C03651=1231.383,135.058,-50.263,-178.039,5.630,148.402
C03652=1231.378,135.308,-50.283,-178.037,5.631,148.401
C03653=1231.373,135.557,-50.304,-178.035,5.632,148.401
C03654=1231.369,135.806,-50.324,-178.032,5.634,148.400
C03655=1231.363,136.055,-50.345,-178.029,5.634,148.400
C03656=1231.359,136.304,-50.365,-178.027,5.635,148.399
C03657=1231.355,136.553,-50.386,-178.024,5.637,148.399
C03658=1231.349,136.802,-50.407,-178.022,5.638,148.398
C03659=1231.345,137.051,-50.427,-178.019,5.638,148.398
C03660=1231.341,137.300,-50.447,-178.017,5.640,148.397
C03661=1231.335,137.549,-50.468,-178.014,5.641,148.397
C03662=1231.331,137.798,-50.489,-178.011,5.643,148.396
C03663=1231.326,138.048,-50.510,-178.009,5.643,148.395
C03664=1231.321,138.297,-50.530,-178.007,5.644,148.395
C03665=1231.316,138.546,-50.551,-178.004,5.646,148.394
C03666=1231.312,138.795,-50.572,-178.001,5.647,148.394
C03667=1231.307,139.044,-50.592,-177.999,5.647,148.393
C03668=1231.302,139.293,-50.613,-177.996,5.649,148.393
C03669=1231.298,139.542,-50.633,-177.994,5.650,148.392
C03670=1231.293,139.791,-50.654,-177.991,5.651,148.392
C03671=1231.288,140.040,-50.675,-177.988,5.652,148.391
C03672=1231.283,140.289,-50.696,-177.986,5.653,148.391
C03673=1231.279,140.539,-50.716,-177.984,5.654,148.390
C03674=1231.274,140.788,-50.737,-177.981,5.656,148.390
C03675=1231.269,141.037,-50.758,-177.978,5.656,148.389
C03676=1231.264,141.287,-50.779,-177.976,5.657,148.389
C03677=1231.260,141.535,-50.800,-177.973,5.659,148.388
C03678=1231.255,141.784,-50.821,-177.971,5.660,148.388
C03679=1231.251,142.033,-50.841,-177.968,5.661,148.387
C03680=1231.245,142.282,-50.862,-177.966,5.662,148.387
C03681=1231.241,142.531,-50.882,-177.963,5.663,148.386
C03682=1231.236,142.781,-50.903,-177.960,5.665,148.386
C03683=1231.231,143.030,-50.924,-177.958,5.665,148.385
C03684=1231.227,143.279,-50.946,-177.956,5.666,148.385
C03685=1231.223,143.528,-50.966,-177.953,5.668,148.384
C03686=1231.217,143.777,-50.987,-177.950,5.669,148.384
C03687=1231.212,144.026,-51.008,-177.947,5.670,148.383
C03688=1231.208,144.275,-51.028,-177.945,5.671,148.383
C03689=1231.203,144.524,-51.050,-177.943,5.672,148.382
C03690=1231.199,144.773,-51.070,-177.940,5.674,148.382
C03691=1231.193,145.022,-51.091,-177.937,5.674,148.381
C03692=1231.189,145.272,-51.112,-177.935,5.676,148.381
C03693=1231.185,145.520,-51.134,-177.932,5.677,148.380
C03694=1231.179,145.770,-51.155,-177.930,5.678,148.380
C03695=1231.175,146.019,-51.175,-177.927,5.680,148.380
C03696=1231.170,146.267,-51.197,-177.925,5.680,148.379
C03697=1231.165,146.517,-51.218,-177.923,5.681,148.379
C03698=1231.161,146.766,-51.239,-177.919,5.683,148.378
C03699=1231.156,147.015,-51.260,-177.917,5.684,148.378
C03700=1231.152,147.264,-51.281,-177.914,5.685,148.377
C03701=1231.147,147.513,-51.302,-177.912,5.686,148.377
C03702=1231.142,147.762,-51.323,-177.909,5.687,148.376
C03703=1231.137,148.011,-51.344,-177.907,5.689,148.376
C03704=1231.133,148.261,-51.365,-177.904,5.689,148.375
C03705=1231.128,148.509,-51.387,-177.902,5.691,148.375
C03706=1231.123,148.758,-51.408,-177.899,5.692,148.374
C03707=1231.119,149.007,-51.429,-177.896,5.694,148.374
C03708=1231.113,149.256,-51.450,-177.894,5.695,148.373
C03709=1231.109,149.506,-51.471,-177.892,5.695,148.372
C03710=1231.105,149.754,-51.492,-177.889,5.697,148.372
C03711=1231.100,150.004,-51.513,-177.886,5.698,148.372
C03712=1231.095,150.252,-51.535,-177.884,5.700,148.371
C03713=1231.090,150.502,-51.556,-177.881,5.700,148.371
C03714=1231.086,150.751,-51.577,-177.879,5.701,148.370
C03715=1231.081,151.000,-51.598,-177.876,5.703,148.370
C03716=1231.076,151.248,-51.620,-177.874,5.704,148.369
C03717=1231.071,151.498,-51.641,-177.871,5.706,148.369
C03718=1231.067,151.747,-51.662,-177.868,5.706,148.368
C03719=1231.062,151.996,-51.683,-177.866,5.708,148.368
C03720=1231.057,152.245,-51.705,-177.863,5.709,148.367
C03721=1231.052,152.494,-51.726,-177.861,5.710,148.367
C03722=1231.048,152.743,-51.748,-177.858,5.712,148.366
C03723=1231.043,152.992,-51.768,-177.856,5.712,148.366
C03724=1231.038,153.241,-51.790,-177.853,5.714,148.365
C03725=1231.034,153.491,-51.811,-177.851,5.715,148.365
C03726=1231.029,153.739,-51.833,-177.848,5.717,148.364
C03727=1231.024,153.988,-51.855,-177.845,5.717,148.364
C03728=1231.020,154.237,-51.875,-177.843,5.719,148.363
C03729=1231.015,154.486,-51.897,-177.841,5.720,148.363
C03730=1231.010,154.736,-51.918,-177.838,5.721,148.362
C03731=1231.005,154.984,-51.940,-177.835,5.723,148.362
C03732=1231.001,155.234,-51.962,-177.833,5.723,148.361
C03733=1230.996,155.483,-51.983,-177.830,5.725,148.361
C03734=1230.991,155.732,-52.004,-177.828,5.726,148.361
C03735=1230.987,155.981,-52.026,-177.825,5.727,148.360
C03736=1230.982,156.230,-52.047,-177.823,5.728,148.360
C03737=1230.977,156.478,-52.069,-177.820,5.730,148.359
C03738=1230.973,156.728,-52.091,-177.817,5.731,148.359
C03739=1230.968,156.977,-52.112,-177.815,5.732,148.358
C03740=1230.963,157.226,-52.133,-177.812,5.733,148.358
C03741=1230.959,157.475,-52.155,-177.810,5.734,148.357
C03742=1230.954,157.724,-52.177,-177.807,5.736,148.357
C03743=1230.949,157.973,-52.198,-177.805,5.737,148.356
C03744=1230.945,158.222,-52.220,-177.802,5.739,148.356
C03745=1230.940,158.471,-52.242,-177.800,5.739,148.355
C03746=1230.935,158.720,-52.263,-177.797,5.741,148.355
C03747=1230.930,158.970,-52.285,-177.794,5.742,148.354
C03748=1230.925,159.218,-52.306,-177.792,5.744,148.354
C03749=1230.921,159.487,-52.330,-177.790,5.745,148.354
C03750=1230.915,159.756,-52.353,-177.786,5.746,148.353
C03751=1230.910,160.025,-52.377,-177.783,5.748,148.352
C03752=1230.906,160.294,-52.400,-177.781,5.749,148.352
C03753=1230.901,160.543,-52.422,-177.778,5.750,148.351
C03754=1230.896,160.792,-52.443,-177.776,5.751,148.351
C03755=1230.892,161.042,-52.465,-177.773,5.753,148.351
C03756=1230.887,161.290,-52.487,-177.771,5.754,148.350
C03757=1230.882,161.539,-52.508,-177.768,5.756,148.350
C03758=1230.878,161.788,-52.530,-177.766,5.757,148.349
C03759=1230.873,162.037,-52.552,-177.763,5.758,148.349
C03760=1230.869,162.286,-52.574,-177.761,5.759,148.348
C03761=1230.864,162.535,-52.596,-177.758,5.761,148.348
C03762=1230.859,162.785,-52.619,-177.755,5.762,148.347
C03763=1230.854,163.033,-52.640,-177.753,5.763,148.347
C03764=1230.849,163.282,-52.662,-177.750,5.764,148.346
C03765=1230.845,163.531,-52.684,-177.748,5.766,148.346
C03766=1230.840,163.780,-52.706,-177.745,5.767,148.346
C03767=1230.836,164.029,-52.728,-177.742,5.768,148.345
C03768=1230.831,164.278,-52.749,-177.740,5.769,148.345
C03769=1230.827,164.527,-52.771,-177.738,5.771,148.344
C03770=1230.822,164.776,-52.793,-177.735,5.772,148.344
C03771=1230.817,165.025,-52.815,-177.732,5.774,148.343
C03772=1230.813,165.274,-52.837,-177.730,5.774,148.343
C03773=1230.808,165.523,-52.859,-177.727,5.776,148.342
C03774=1230.803,165.772,-52.881,-177.725,5.777,148.342
C03775=1230.798,166.021,-52.903,-177.722,5.779,148.341
C03776=1230.794,166.270,-52.925,-177.720,5.780,148.341
C03777=1230.789,166.519,-52.947,-177.717,5.782,148.340
C03778=1230.784,166.768,-52.969,-177.715,5.782,148.340
C03779=1230.779,167.018,-52.991,-177.712,5.784,148.340
C03780=1230.775,167.266,-53.013,-177.710,5.785,148.339
C03781=1230.770,167.516,-53.035,-177.707,5.787,148.339
C03782=1230.766,167.764,-53.057,-177.705,5.788,148.338
C03783=1230.761,168.013,-53.079,-177.702,5.789,148.338
C03784=1230.756,168.262,-53.102,-177.699,5.791,148.337
C03785=1230.752,168.511,-53.124,-177.697,5.792,148.337
C03786=1230.747,168.760,-53.145,-177.694,5.794,148.336
C03787=1230.742,169.009,-53.167,-177.691,5.794,148.336
C03788=1230.738,169.257,-53.190,-177.689,5.796,148.335
C03789=1230.733,169.507,-53.213,-177.687,5.797,148.335
C03790=1230.728,169.756,-53.234,-177.684,5.799,148.335
C03791=1230.724,170.005,-53.256,-177.681,5.800,148.334
C03792=1230.719,170.254,-53.278,-177.679,5.802,148.334
C03793=1230.714,170.503,-53.301,-177.676,5.802,148.333
C03794=1230.710,170.752,-53.323,-177.674,5.804,148.333
C03795=1230.705,171.001,-53.345,-177.671,5.805,148.332
C03796=1230.700,171.250,-53.368,-177.669,5.807,148.332
C03797=1230.695,171.498,-53.390,-177.666,5.808,148.331
C03798=1230.691,171.748,-53.412,-177.664,5.809,148.331
C03799=1230.686,171.997,-53.434,-177.661,5.811,148.331
C03800=1230.682,172.245,-53.457,-177.658,5.812,148.330
C03801=1230.677,172.495,-53.479,-177.656,5.814,148.330
C03802=1230.672,172.743,-53.501,-177.654,5.815,148.329
C03803=1230.668,172.992,-53.524,-177.650,5.816,148.329
C03804=1230.663,173.241,-53.546,-177.648,5.817,148.328
C03805=1230.658,173.491,-53.569,-177.646,5.819,148.328
C03806=1230.654,173.739,-53.591,-177.643,5.821,148.327
C03807=1230.649,173.988,-53.613,-177.640,5.822,148.327
C03808=1230.644,174.238,-53.636,-177.638,5.823,148.327
C03809=1230.640,174.486,-53.658,-177.636,5.824,148.326
C03810=1230.635,174.735,-53.680,-177.633,5.826,148.326
C03811=1230.631,174.984,-53.703,-177.630,5.827,148.325
C03812=1230.626,175.233,-53.725,-177.628,5.829,148.325
C03813=1230.621,175.482,-53.749,-177.625,5.830,148.324
C03814=1230.617,175.731,-53.771,-177.623,5.831,148.324
C03815=1230.612,175.980,-53.792,-177.620,5.833,148.324
C03816=1230.607,176.229,-53.816,-177.618,5.834,148.323
C03817=1230.603,176.478,-53.838,-177.615,5.836,148.323
C03818=1230.598,176.726,-53.861,-177.613,5.837,148.322
C03819=1230.593,176.976,-53.883,-177.610,5.839,148.322
C03820=1230.589,177.225,-53.906,-177.607,5.840,148.321
C03821=1230.584,177.473,-53.928,-177.605,5.841,148.321
C03822=1230.579,177.722,-53.951,-177.602,5.843,148.321
C03823=1230.575,177.971,-53.974,-177.600,5.844,148.320
C03824=1230.570,178.220,-53.996,-177.597,5.845,148.320
C03825=1230.565,178.469,-54.019,-177.594,5.847,148.319
C03826=1230.561,178.718,-54.041,-177.592,5.848,148.319
C03827=1230.556,178.967,-54.064,-177.589,5.850,148.318
C03828=1230.552,179.216,-54.086,-177.587,5.851,148.318
C03829=1230.547,179.465,-54.109,-177.584,5.853,148.318
C03830=1230.543,179.714,-54.132,-177.582,5.854,148.317
C03831=1230.537,179.963,-54.154,-177.579,5.855,148.317
C03832=1230.533,180.212,-54.178,-177.576,5.857,148.316
C03833=1230.528,180.461,-54.200,-177.574,5.858,148.316
C03834=1230.524,180.710,-54.223,-177.572,5.860,148.316
C03835=1230.519,180.958,-54.246,-177.569,5.861,148.315
C03836=1230.514,181.208,-54.268,-177.566,5.862,148.315
C03837=1230.510,181.456,-54.291,-177.564,5.864,148.314
C03838=1230.505,181.705,-54.314,-177.562,5.865,148.314
C03839=1230.501,181.953,-54.337,-177.559,5.867,148.313
C03840=1230.496,182.203,-54.359,-177.556,5.869,148.313
C03841=1230.491,182.452,-54.383,-177.554,5.870,148.313
C03842=1230.487,182.701,-54.405,-177.551,5.871,148.312
C03843=1230.482,182.950,-54.428,-177.548,5.873,148.312
C03844=1230.478,183.198,-54.451,-177.546,5.874,148.311
C03845=1230.473,183.447,-54.474,-177.543,5.876,148.311
C03846=1230.468,183.697,-54.497,-177.541,5.877,148.311
C03847=1230.464,183.945,-54.520,-177.538,5.878,148.310
C03848=1230.459,184.194,-54.542,-177.535,5.880,148.310
C03849=1230.454,184.443,-54.566,-177.533,5.881,148.309
C03850=1230.450,184.692,-54.588,-177.531,5.883,148.309
C03851=1230.445,184.941,-54.612,-177.528,5.885,148.308
C03852=1230.441,185.190,-54.635,-177.525,5.886,148.308
C03853=1230.436,185.459,-54.660,-177.523,5.887,148.308
C03854=1230.431,185.729,-54.685,-177.520,5.889,148.307
C03855=1230.425,185.999,-54.710,-177.517,5.891,148.307
C03856=1230.421,186.268,-54.734,-177.514,5.893,148.306
C03857=1230.416,186.517,-54.757,-177.512,5.893,148.306
C03858=1230.411,186.767,-54.781,-177.509,5.895,148.305
C03859=1230.407,187.015,-54.803,-177.507,5.897,148.305
C03860=1230.402,187.264,-54.827,-177.504,5.898,148.305
C03861=1230.397,187.513,-54.850,-177.501,5.900,148.304
C03862=1230.392,187.762,-54.873,-177.499,5.901,148.304
C03863=1230.388,188.011,-54.895,-177.497,5.902,148.303
C03864=1230.384,188.260,-54.919,-177.494,5.904,148.303
C03865=1230.379,188.509,-54.942,-177.492,5.905,148.303
C03866=1230.374,188.757,-54.965,-177.489,5.907,148.302
C03867=1230.370,189.006,-54.988,-177.486,5.909,148.302
C03868=1230.365,189.255,-55.011,-177.484,5.910,148.301
C03869=1230.360,189.504,-55.035,-177.481,5.912,148.301
C03870=1230.356,189.753,-55.058,-177.479,5.913,148.301
C03871=1230.351,190.002,-55.081,-177.476,5.914,148.300
C03872=1230.347,190.251,-55.104,-177.474,5.916,148.300
C03873=1230.342,190.500,-55.127,-177.471,5.918,148.299
C03874=1230.338,190.748,-55.151,-177.469,5.919,148.299
C03875=1230.333,190.997,-55.174,-177.466,5.921,148.299
C03876=1230.328,191.246,-55.198,-177.463,5.922,148.298
C03877=1230.323,191.495,-55.221,-177.460,5.924,148.298
C03878=1230.319,191.743,-55.244,-177.458,5.925,148.297
C03879=1230.315,191.993,-55.267,-177.456,5.927,148.297
C03880=1230.310,192.242,-55.291,-177.453,5.929,148.297
C03881=1230.305,192.491,-55.314,-177.450,5.929,148.296
C03882=1230.301,192.740,-55.337,-177.448,5.931,148.296
C03883=1230.296,192.988,-55.361,-177.445,5.933,148.295
C03884=1230.291,193.237,-55.385,-177.443,5.934,148.295
C03885=1230.287,193.486,-55.408,-177.440,5.936,148.295
C03886=1230.283,193.735,-55.431,-177.438,5.938,148.294
C03887=1230.278,193.984,-55.454,-177.435,5.938,148.294
C03888=1230.273,194.233,-55.478,-177.433,5.940,148.293
C03889=1230.269,194.481,-55.502,-177.430,5.942,148.293
C03890=1230.264,194.730,-55.525,-177.428,5.943,148.293
C03891=1230.260,194.979,-55.548,-177.425,5.945,148.292
C03892=1230.255,195.228,-55.572,-177.423,5.947,148.292
C03893=1230.250,195.477,-55.596,-177.419,5.948,148.291
C03894=1230.246,195.726,-55.619,-177.417,5.949,148.291
C03895=1230.241,195.975,-55.643,-177.415,5.951,148.291
C03896=1230.236,196.224,-55.666,-177.412,5.953,148.290
C03897=1230.232,196.472,-55.690,-177.410,5.954,148.290
C03898=1230.227,196.721,-55.713,-177.407,5.956,148.289
C03899=1230.223,196.970,-55.737,-177.404,5.958,148.289
C03900=1230.218,197.219,-55.761,-177.402,5.959,148.289
C03901=1230.213,197.468,-55.784,-177.400,5.960,148.288
C03902=1230.209,197.717,-55.808,-177.397,5.962,148.288
C03903=1230.204,197.965,-55.832,-177.394,5.964,148.288
C03904=1230.200,198.214,-55.855,-177.392,5.965,148.287
C03905=1230.195,198.463,-55.879,-177.389,5.967,148.287
C03906=1230.191,198.712,-55.902,-177.386,5.969,148.286
C03907=1230.186,198.961,-55.926,-177.384,5.970,148.286
C03908=1230.182,199.209,-55.950,-177.382,5.971,148.286
C03909=1230.177,199.458,-55.973,-177.379,5.973,148.285
C03910=1230.172,199.707,-55.997,-177.376,5.975,148.285
C03911=1230.168,199.956,-56.021,-177.374,5.976,148.284
C03912=1230.163,200.205,-56.044,-177.371,5.978,148.284
C03913=1230.158,200.453,-56.069,-177.369,5.980,148.284
C03914=1230.153,200.702,-56.092,-177.366,5.981,148.283
C03915=1230.149,200.951,-56.116,-177.364,5.982,148.283
C03916=1230.144,201.200,-56.139,-177.361,5.984,148.283
C03917=1230.140,201.449,-56.164,-177.359,5.986,148.282
C03918=1230.136,201.698,-56.187,-177.356,5.988,148.282
C03919=1230.131,201.946,-56.211,-177.353,5.989,148.281
C03920=1230.126,202.196,-56.235,-177.351,5.991,148.281
C03921=1230.121,202.444,-56.259,-177.348,5.992,148.281
C03922=1230.117,202.693,-56.283,-177.345,5.994,148.280
C03923=1230.112,202.942,-56.307,-177.343,5.995,148.280
C03924=1230.108,203.190,-56.331,-177.341,5.997,148.280
C03925=1230.103,203.439,-56.354,-177.338,5.999,148.279
C03926=1230.099,203.688,-56.379,-177.335,6.001,148.279
C03927=1230.094,203.937,-56.403,-177.333,6.002,148.278
C03928=1230.090,204.186,-56.427,-177.330,6.003,148.278
C03929=1230.085,204.434,-56.451,-177.328,6.005,148.278
C03930=1230.080,204.683,-56.474,-177.325,6.007,148.277
C03931=1230.076,204.932,-56.498,-177.323,6.008,148.277
C03932=1230.071,205.181,-56.523,-177.320,6.010,148.277
C03933=1230.067,205.430,-56.547,-177.318,6.012,148.276
C03934=1230.062,205.679,-56.571,-177.315,6.014,148.276
C03935=1230.058,205.927,-56.595,-177.312,6.016,148.276
C03936=1230.053,206.176,-56.619,-177.310,6.017,148.275
C03937=1230.048,206.425,-56.643,-177.307,6.018,148.275
C03938=1230.044,206.674,-56.667,-177.305,6.020,148.274
C03939=1230.040,206.922,-56.691,-177.302,6.022,148.274
C03940=1230.035,207.172,-56.715,-177.300,6.023,148.274
C03941=1230.030,207.420,-56.739,-177.297,6.025,148.273
C03942=1230.026,207.669,-56.763,-177.295,6.027,148.273
C03943=1230.021,207.917,-56.788,-177.292,6.028,148.273
C03944=1230.017,208.167,-56.812,-177.289,6.030,148.272
C03945=1230.012,208.415,-56.836,-177.287,6.031,148.272
C03946=1230.008,208.664,-56.860,-177.285,6.033,148.271
C03947=1230.003,208.913,-56.885,-177.282,6.035,148.271
C03948=1229.999,209.162,-56.909,-177.279,6.037,148.271
C03949=1229.994,209.410,-56.934,-177.276,6.038,148.270
C03950=1229.989,209.659,-56.957,-177.274,6.039,148.270
C03951=1229.985,209.908,-56.981,-177.272,6.041,148.270
C03952=1229.979,210.157,-57.006,-177.269,6.043,148.269
C03953=1229.976,210.406,-57.030,-177.266,6.045,148.269
C03954=1229.971,210.654,-57.054,-177.264,6.047,148.269
C03955=1229.966,210.903,-57.079,-177.262,6.048,148.268
C03956=1229.962,211.151,-57.103,-177.259,6.050,148.268
C03957=1229.957,211.423,-57.129,-177.256,6.051,148.267
C03958=1229.952,211.693,-57.156,-177.253,6.053,148.267
C03959=1229.947,211.963,-57.183,-177.251,6.055,148.267
C03960=1229.942,212.233,-57.209,-177.248,6.057,148.266
C03961=1229.938,212.482,-57.234,-177.245,6.059,148.266
C03962=1229.933,212.731,-57.258,-177.243,6.061,148.266
C03963=1229.928,212.979,-57.283,-177.240,6.063,148.265
C03964=1229.924,213.229,-57.307,-177.237,6.064,148.265
C03965=1229.919,213.477,-57.332,-177.235,6.065,148.264
C03966=1229.915,213.726,-57.356,-177.232,6.067,148.264
C03967=1229.910,213.974,-57.381,-177.230,6.069,148.264
C03968=1229.906,214.224,-57.405,-177.227,6.071,148.263
C03969=1229.901,214.472,-57.430,-177.224,6.073,148.263
C03970=1229.896,214.721,-57.454,-177.222,6.074,148.263
C03971=1229.892,214.970,-57.479,-177.220,6.075,148.262
C03972=1229.887,215.219,-57.503,-177.217,6.077,148.262
C03973=1229.882,215.467,-57.528,-177.214,6.079,148.262
C03974=1229.879,215.716,-57.552,-177.212,6.081,148.261
C03975=1229.873,215.965,-57.577,-177.209,6.083,148.261
C03976=1229.869,216.213,-57.601,-177.207,6.085,148.261
C03977=1229.865,216.462,-57.626,-177.204,6.086,148.260
C03978=1229.860,216.711,-57.651,-177.202,6.088,148.260
C03979=1229.856,216.960,-57.676,-177.199,6.089,148.260
C03980=1229.851,217.209,-57.700,-177.197,6.091,148.259
C03981=1229.846,217.457,-57.724,-177.194,6.093,148.259
C03982=1229.842,217.706,-57.750,-177.191,6.095,148.259
C03983=1229.838,217.955,-57.774,-177.189,6.097,148.258
C03984=1229.833,218.203,-57.799,-177.187,6.098,148.258
C03985=1229.829,218.452,-57.823,-177.184,6.100,148.258
C03986=1229.824,218.701,-57.848,-177.181,6.102,148.257
C03987=1229.819,218.950,-57.874,-177.179,6.104,148.257
C03988=1229.815,219.198,-57.898,-177.176,6.105,148.257
C03989=1229.810,219.447,-57.922,-177.173,6.107,148.256
C03990=1229.806,219.696,-57.948,-177.171,6.108,148.256
C03991=1229.801,219.944,-57.972,-177.168,6.110,148.255
C03992=1229.797,220.194,-57.997,-177.166,6.112,148.255
C03993=1229.792,220.442,-58.021,-177.163,6.114,148.255
C03994=1229.788,220.691,-58.047,-177.160,6.116,148.254
C03995=1229.783,220.940,-58.072,-177.158,6.117,148.254
C03996=1229.779,221.188,-58.096,-177.155,6.119,148.254
C03997=1229.774,221.437,-58.122,-177.153,6.120,148.253
C03998=1229.769,221.686,-58.146,-177.150,6.122,148.253
C03999=1229.766,221.934,-58.171,-177.148,6.124,148.253
C04000=1229.761,222.183,-58.196,-177.145,6.126,148.252
C04001=1229.756,222.432,-58.221,-177.143,6.128,148.252
C04002=1229.751,222.680,-58.247,-177.140,6.130,148.252
C04003=1229.747,222.929,-58.271,-177.137,6.131,148.251
C04004=1229.743,223.178,-58.296,-177.135,6.134,148.251
C04005=1229.738,223.427,-58.321,-177.133,6.135,148.251
C04006=1229.733,223.676,-58.346,-177.130,6.137,148.251
C04007=1229.730,223.924,-58.371,-177.128,6.138,148.250
C04008=1229.724,224.173,-58.396,-177.125,6.140,148.250
C04009=1229.720,224.421,-58.421,-177.123,6.142,148.250
C04010=1229.715,224.670,-58.446,-177.120,6.144,148.249
C04011=1229.711,224.918,-58.471,-177.117,6.146,148.249
C04012=1229.706,225.168,-58.496,-177.115,6.147,148.249
C04013=1229.702,225.416,-58.522,-177.113,6.149,148.248
C04014=1229.697,225.665,-58.547,-177.110,6.151,148.248
C04015=1229.693,225.914,-58.572,-177.107,6.153,148.248
C04016=1229.689,226.162,-58.597,-177.105,6.154,148.247
C04017=1229.684,226.411,-58.622,-177.102,6.156,148.247
C04018=1229.679,226.659,-58.647,-177.100,6.158,148.247
C04019=1229.675,226.909,-58.673,-177.097,6.160,148.246
C04020=1229.670,227.157,-58.698,-177.094,6.162,148.246
C04021=1229.665,227.406,-58.723,-177.092,6.163,148.246
C04022=1229.661,227.654,-58.748,-177.090,6.165,148.245
C04023=1229.657,227.903,-58.773,-177.087,6.167,148.245
C04024=1229.652,228.152,-58.798,-177.084,6.169,148.245
C04025=1229.648,228.400,-58.824,-177.082,6.170,148.244
C04026=1229.644,228.649,-58.850,-177.079,6.172,148.244
C04027=1229.638,228.898,-58.874,-177.077,6.174,148.244
C04028=1229.634,229.147,-58.900,-177.074,6.176,148.244
C04029=1229.629,229.395,-58.925,-177.072,6.178,148.243
C04030=1229.625,229.644,-58.951,-177.070,6.179,148.243
C04031=1229.620,229.892,-58.976,-177.067,6.181,148.243
C04032=1229.616,230.141,-59.002,-177.064,6.183,148.242
C04033=1229.612,230.390,-59.027,-177.062,6.185,148.242
C04034=1229.606,230.639,-59.052,-177.059,6.187,148.242
C04035=1229.603,230.887,-59.077,-177.057,6.189,148.241
C04036=1229.598,231.135,-59.103,-177.054,6.191,148.241
C04037=1229.594,231.384,-59.128,-177.051,6.192,148.241
C04038=1229.590,231.633,-59.154,-177.049,6.194,148.240
C04039=1229.585,231.882,-59.179,-177.046,6.196,148.240
C04040=1229.580,232.130,-59.205,-177.044,6.197,148.240
C04041=1229.576,232.379,-59.230,-177.041,6.199,148.239
C04042=1229.571,232.627,-59.256,-177.039,6.201,148.239
C04043=1229.567,232.876,-59.281,-177.037,6.203,148.239
C04044=1229.563,233.125,-59.307,-177.034,6.205,148.239
C04045=1229.558,233.374,-59.332,-177.031,6.207,148.238
C04046=1229.553,233.623,-59.358,-177.029,6.209,148.238
C04047=1229.549,233.872,-59.384,-177.026,6.211,148.238
C04048=1229.544,234.120,-59.409,-177.024,6.213,148.237
C04049=1229.539,234.368,-59.435,-177.021,6.214,148.237
C04050=1229.535,234.617,-59.461,-177.018,6.216,148.237
C04051=1229.530,234.865,-59.486,-177.016,6.217,148.236
C04052=1229.526,235.114,-59.512,-177.014,6.219,148.236
C04053=1229.522,235.363,-59.538,-177.012,6.221,148.236
C04054=1229.517,235.611,-59.563,-177.009,6.223,148.236
C04055=1229.513,235.860,-59.589,-177.006,6.225,148.235
C04056=1229.509,236.109,-59.615,-177.004,6.227,148.235
C04057=1229.504,236.357,-59.640,-177.001,6.229,148.235
C04058=1229.499,236.606,-59.666,-176.998,6.231,148.234
C04059=1229.495,236.855,-59.692,-176.996,6.233,148.234
C04060=1229.490,237.104,-59.718,-176.994,6.235,148.234
C04061=1229.485,237.375,-59.745,-176.991,6.236,148.234
C04062=1229.480,237.647,-59.774,-176.988,6.238,148.233
C04063=1229.476,237.917,-59.802,-176.985,6.240,148.233
C04064=1229.471,238.189,-59.830,-176.982,6.243,148.233
C04065=1229.467,238.438,-59.856,-176.980,6.245,148.232
C04066=1229.462,238.686,-59.881,-176.977,6.247,148.232
C04067=1229.457,238.935,-59.907,-176.975,6.248,148.232
C04068=1229.453,239.184,-59.933,-176.973,6.250,148.232
C04069=1229.449,239.432,-59.960,-176.970,6.252,148.231
C04070=1229.444,239.680,-59.985,-176.968,6.254,148.231
C04071=1229.440,239.929,-60.011,-176.965,6.255,148.231
C04072=1229.435,240.178,-60.037,-176.962,6.257,148.230
C04073=1229.430,240.427,-60.063,-176.960,6.260,148.230
C04074=1229.426,240.675,-60.088,-176.958,6.261,148.230
C04075=1229.422,240.923,-60.115,-176.955,6.263,148.230
C04076=1229.417,241.172,-60.141,-176.952,6.265,148.229
C04077=1229.412,241.421,-60.167,-176.950,6.267,148.229
C04078=1229.408,241.670,-60.193,-176.947,6.269,148.229
C04079=1229.404,241.917,-60.219,-176.945,6.271,148.229
C04080=1229.399,242.167,-60.245,-176.942,6.273,148.228
C04081=1229.395,242.415,-60.271,-176.940,6.275,148.228
C04082=1229.390,242.664,-60.297,-176.937,6.277,148.228
C04083=1229.386,242.913,-60.324,-176.935,6.279,148.227
C04084=1229.381,243.161,-60.349,-176.932,6.281,148.227
C04085=1229.377,243.410,-60.375,-176.930,6.283,148.227
C04086=1229.372,243.658,-60.402,-176.927,6.285,148.227
C04087=1229.368,243.907,-60.428,-176.925,6.287,148.226
C04088=1229.364,244.156,-60.453,-176.922,6.288,148.226
C04089=1229.359,244.404,-60.480,-176.919,6.290,148.226
C04090=1229.354,244.652,-60.506,-176.918,6.292,148.226
C04091=1229.350,244.901,-60.531,-176.915,6.294,148.225
C04092=1229.345,245.150,-60.559,-176.913,6.295,148.225
C04093=1229.341,245.398,-60.584,-176.910,6.297,148.225
C04094=1229.337,245.647,-60.610,-176.907,6.299,148.224
C04095=1229.332,245.896,-60.637,-176.905,6.301,148.224
C04096=1229.328,246.144,-60.663,-176.903,6.303,148.224
C04097=1229.323,246.393,-60.690,-176.900,6.305,148.224
C04098=1229.318,246.641,-60.715,-176.897,6.307,148.223
C04099=1229.314,246.890,-60.742,-176.895,6.309,148.223
C04100=1229.309,247.138,-60.768,-176.893,6.311,148.223
C04101=1229.306,247.387,-60.795,-176.890,6.313,148.223
C04102=1229.301,247.636,-60.821,-176.887,6.315,148.222
C04103=1229.297,247.884,-60.847,-176.885,6.317,148.222
C04104=1229.292,248.133,-60.874,-176.882,6.319,148.222
C04105=1229.288,248.381,-60.900,-176.880,6.321,148.222
C04106=1229.283,248.630,-60.927,-176.877,6.323,148.221
C04107=1229.279,248.878,-60.953,-176.875,6.325,148.221
C04108=1229.274,249.128,-60.979,-176.872,6.326,148.221
C04109=1229.269,249.375,-61.005,-176.870,6.329,148.221
C04110=1229.264,249.624,-61.032,-176.867,6.331,148.220
C04111=1229.261,249.872,-61.058,-176.865,6.332,148.220
C04112=1229.256,250.121,-61.085,-176.862,6.334,148.220
C04113=1229.252,250.370,-61.111,-176.860,6.336,148.219
C04114=1229.247,250.618,-61.138,-176.858,6.338,148.219
C04115=1229.243,250.867,-61.164,-176.855,6.340,148.219
C04116=1229.238,251.115,-61.191,-176.852,6.342,148.219
C04117=1229.234,251.364,-61.217,-176.850,6.344,148.218
C04118=1229.229,251.613,-61.244,-176.848,6.346,148.218
C04119=1229.225,251.861,-61.270,-176.845,6.348,148.218
C04120=1229.221,252.109,-61.297,-176.842,6.350,148.218
C04121=1229.216,252.358,-61.324,-176.840,6.352,148.217
C04122=1229.212,252.607,-61.350,-176.838,6.354,148.217
C04123=1229.207,252.855,-61.377,-176.835,6.356,148.217
C04124=1229.203,253.103,-61.404,-176.832,6.358,148.217
C04125=1229.198,253.353,-61.430,-176.830,6.360,148.216
C04126=1229.194,253.601,-61.457,-176.828,6.362,148.216
C04127=1229.190,253.849,-61.484,-176.825,6.364,148.216
C04128=1229.185,254.098,-61.511,-176.822,6.366,148.216
C04129=1229.180,254.346,-61.538,-176.820,6.368,148.215
C04130=1229.176,254.595,-61.563,-176.817,6.371,148.215
C04131=1229.171,254.843,-61.590,-176.815,6.373,148.215
C04132=1229.168,255.092,-61.617,-176.812,6.374,148.215
C04133=1229.163,255.340,-61.644,-176.810,6.377,148.215
C04134=1229.158,255.589,-61.671,-176.807,6.379,148.214
C04135=1229.153,255.838,-61.697,-176.805,6.380,148.214
C04136=1229.149,256.086,-61.724,-176.803,6.383,148.214
C04137=1229.145,256.334,-61.751,-176.800,6.385,148.214
C04138=1229.141,256.584,-61.778,-176.797,6.386,148.213
C04139=1229.137,256.832,-61.805,-176.795,6.388,148.213
C04140=1229.132,257.080,-61.832,-176.793,6.391,148.213
C04141=1229.127,257.329,-61.859,-176.790,6.392,148.213
C04142=1229.123,257.577,-61.886,-176.787,6.394,148.212
C04143=1229.119,257.826,-61.912,-176.785,6.397,148.212
C04144=1229.114,258.074,-61.940,-176.783,6.398,148.212
C04145=1229.110,258.323,-61.967,-176.780,6.400,148.212
C04146=1229.105,258.571,-61.994,-176.778,6.402,148.211
C04147=1229.101,258.819,-62.020,-176.775,6.404,148.211
C04148=1229.096,259.068,-62.047,-176.773,6.406,148.211
C04149=1229.092,259.317,-62.075,-176.771,6.408,148.211
C04150=1229.088,259.565,-62.102,-176.768,6.410,148.210
C04151=1229.084,259.814,-62.128,-176.765,6.412,148.210
C04152=1229.079,260.062,-62.155,-176.762,6.415,148.210
C04153=1229.074,260.311,-62.182,-176.760,6.417,148.210
C04154=1229.070,260.559,-62.209,-176.757,6.419,148.210
C04155=1229.065,260.808,-62.236,-176.755,6.421,148.209
C04156=1229.060,261.056,-62.263,-176.753,6.423,148.209
C04157=1229.057,261.305,-62.290,-176.750,6.425,148.209
C04158=1229.052,261.553,-62.317,-176.748,6.427,148.209
C04159=1229.048,261.802,-62.344,-176.745,6.429,148.208
C04160=1229.043,262.050,-62.371,-176.743,6.431,148.208
C04161=1229.039,262.298,-62.399,-176.741,6.433,148.208
C04162=1229.034,262.547,-62.426,-176.738,6.435,148.208
C04163=1229.030,262.796,-62.454,-176.735,6.437,148.207
C04164=1229.025,263.044,-62.481,-176.733,6.439,148.207
C04165=1229.021,263.317,-62.511,-176.730,6.442,148.207
C04166=1229.016,263.589,-62.540,-176.728,6.444,148.207
C04167=1229.011,263.862,-62.571,-176.724,6.447,148.207
C04168=1229.006,264.135,-62.600,-176.722,6.448,148.206
C04169=1229.002,264.383,-62.627,-176.720,6.451,148.206
C04170=1228.998,264.632,-62.655,-176.717,6.453,148.206
C04171=1228.993,264.880,-62.682,-176.715,6.455,148.206
C04172=1228.988,265.129,-62.709,-176.712,6.457,148.206
C04173=1228.984,265.377,-62.737,-176.710,6.459,148.205
C04174=1228.979,265.625,-62.764,-176.708,6.461,148.205
C04175=1228.975,265.874,-62.791,-176.705,6.464,148.205
C04176=1228.971,266.122,-62.819,-176.702,6.465,148.205
C04177=1228.966,266.371,-62.846,-176.700,6.468,148.205
C04178=1228.962,266.619,-62.873,-176.697,6.470,148.204
C04179=1228.958,266.868,-62.901,-176.695,6.472,148.204
C04180=1228.953,267.116,-62.928,-176.692,6.474,148.204
C04181=1228.949,267.365,-62.955,-176.690,6.476,148.204
C04182=1228.944,267.613,-62.983,-176.688,6.478,148.204
C04183=1228.940,267.862,-63.011,-176.685,6.480,148.203
C04184=1228.936,268.110,-63.038,-176.683,6.483,148.203
C04185=1228.931,268.358,-63.065,-176.680,6.485,148.203
C04186=1228.927,268.607,-63.092,-176.677,6.486,148.203
C04187=1228.923,268.855,-63.121,-176.675,6.489,148.203
C04188=1228.918,269.104,-63.148,-176.673,6.491,148.202
C04189=1228.914,269.352,-63.175,-176.670,6.493,148.202
C04190=1228.909,269.601,-63.203,-176.668,6.495,148.202
C04191=1228.905,269.849,-63.231,-176.666,6.497,148.202
C04192=1228.900,270.097,-63.258,-176.663,6.499,148.201
C04193=1228.896,270.345,-63.286,-176.660,6.501,148.201
C04194=1228.892,270.595,-63.313,-176.658,6.504,148.201
C04195=1228.887,270.842,-63.341,-176.655,6.506,148.201
C04196=1228.883,271.091,-63.368,-176.653,6.508,148.201
C04197=1228.879,271.339,-63.396,-176.651,6.510,148.200
C04198=1228.874,271.588,-63.424,-176.648,6.512,148.200
C04199=1228.869,271.836,-63.452,-176.646,6.514,148.200
C04200=1228.865,272.085,-63.479,-176.644,6.516,148.200
C04201=1228.861,272.333,-63.507,-176.641,6.519,148.200
C04202=1228.856,272.581,-63.535,-176.638,6.521,148.200
C04203=1228.852,272.830,-63.562,-176.636,6.523,148.199
C04204=1228.847,273.079,-63.591,-176.633,6.525,148.199
C04205=1228.844,273.327,-63.619,-176.631,6.527,148.199
C04206=1228.839,273.576,-63.646,-176.629,6.529,148.199
C04207=1228.835,273.823,-63.674,-176.626,6.531,148.199
C04208=1228.830,274.073,-63.701,-176.623,6.534,148.198
C04209=1228.825,274.321,-63.729,-176.621,6.536,148.198
C04210=1228.821,274.569,-63.757,-176.619,6.538,148.198
C04211=1228.817,274.817,-63.785,-176.616,6.540,148.198
C04212=1228.813,275.066,-63.812,-176.614,6.542,148.198
C04213=1228.808,275.315,-63.841,-176.612,6.544,148.198
C04214=1228.804,275.563,-63.869,-176.609,6.547,148.197
C04215=1228.799,275.810,-63.897,-176.606,6.549,148.197
C04216=1228.795,276.060,-63.924,-176.604,6.551,148.197
C04217=1228.790,276.308,-63.952,-176.602,6.553,148.197
C04218=1228.787,276.556,-63.981,-176.599,6.555,148.197
C04219=1228.782,276.804,-64.008,-176.597,6.557,148.197
C04220=1228.777,277.053,-64.036,-176.594,6.559,148.196
C04221=1228.773,277.302,-64.064,-176.592,6.562,148.196
C04222=1228.769,277.550,-64.092,-176.589,6.564,148.196
C04223=1228.764,277.798,-64.121,-176.587,6.566,148.196
C04224=1228.760,278.046,-64.149,-176.584,6.568,148.196
C04225=1228.756,278.295,-64.177,-176.582,6.571,148.196
C04226=1228.751,278.543,-64.205,-176.580,6.572,148.195
C04227=1228.747,278.792,-64.232,-176.577,6.576,148.195
C04228=1228.743,279.040,-64.260,-176.575,6.577,148.195
C04229=1228.738,279.289,-64.289,-176.572,6.580,148.195
C04230=1228.734,279.537,-64.317,-176.570,6.582,148.195
C04231=1228.730,279.785,-64.345,-176.568,6.584,148.195
C04232=1228.725,280.034,-64.373,-176.565,6.587,148.195
C04233=1228.721,280.282,-64.401,-176.562,6.589,148.194
C04234=1228.716,280.530,-64.430,-176.560,6.591,148.194
C04235=1228.712,280.779,-64.458,-176.558,6.593,148.194
C04236=1228.707,281.027,-64.486,-176.556,6.595,148.194
C04237=1228.703,281.276,-64.514,-176.553,6.597,148.194
C04238=1228.699,281.524,-64.542,-176.550,6.600,148.194
C04239=1228.695,281.773,-64.571,-176.548,6.602,148.193
C04240=1228.690,282.020,-64.599,-176.546,6.604,148.193
C04241=1228.686,282.269,-64.627,-176.544,6.606,148.193
C04242=1228.681,282.517,-64.655,-176.541,6.608,148.193
C04243=1228.677,282.766,-64.684,-176.538,6.611,148.193
C04244=1228.673,283.014,-64.712,-176.536,6.613,148.193
C04245=1228.668,283.263,-64.740,-176.534,6.615,148.192
C04246=1228.664,283.511,-64.768,-176.531,6.618,148.192
C04247=1228.660,283.759,-64.798,-176.529,6.619,148.192
C04248=1228.655,284.007,-64.825,-176.526,6.623,148.192
C04249=1228.651,284.256,-64.854,-176.524,6.624,148.192
C04250=1228.646,284.504,-64.882,-176.521,6.627,148.192
C04251=1228.642,284.752,-64.911,-176.519,6.629,148.192
C04252=1228.638,285.001,-64.939,-176.517,6.631,148.191
C04253=1228.633,285.249,-64.967,-176.514,6.634,148.191
C04254=1228.629,285.497,-64.997,-176.512,6.636,148.191
C04255=1228.625,285.745,-65.024,-176.509,6.638,148.191
C04256=1228.620,285.994,-65.053,-176.507,6.640,148.191
C04257=1228.616,286.243,-65.081,-176.505,6.642,148.191
C04258=1228.612,286.490,-65.110,-176.502,6.645,148.191
C04259=1228.608,286.739,-65.139,-176.500,6.647,148.191
C04260=1228.603,286.987,-65.167,-176.497,6.649,148.190
C04261=1228.598,287.236,-65.196,-176.495,6.651,148.190
C04262=1228.595,287.484,-65.225,-176.493,6.654,148.190
C04263=1228.590,287.732,-65.253,-176.490,6.656,148.190
C04264=1228.585,287.981,-65.282,-176.488,6.659,148.190
C04265=1228.581,288.228,-65.310,-176.486,6.661,148.190
C04266=1228.577,288.477,-65.339,-176.483,6.663,148.189
C04267=1228.572,288.726,-65.368,-176.481,6.666,148.189
C04268=1228.568,288.973,-65.396,-176.478,6.668,148.189
C04269=1228.563,289.248,-65.428,-176.476,6.670,148.189
C04270=1228.559,289.522,-65.459,-176.473,6.673,148.189
C04271=1228.554,289.796,-65.491,-176.471,6.675,148.189
C04272=1228.549,290.071,-65.523,-176.468,6.678,148.189
C04273=1228.544,290.318,-65.552,-176.465,6.680,148.189
C04274=1228.540,290.567,-65.580,-176.463,6.683,148.189
C04275=1228.536,290.815,-65.609,-176.461,6.685,148.188
C04276=1228.531,291.063,-65.638,-176.458,6.687,148.188
C04277=1228.528,291.311,-65.667,-176.456,6.689,148.188
C04278=1228.523,291.560,-65.695,-176.454,6.691,148.188
C04279=1228.518,291.808,-65.724,-176.451,6.694,148.188
C04280=1228.514,292.057,-65.753,-176.449,6.696,148.188
C04281=1228.510,292.305,-65.782,-176.446,6.699,148.188
C04282=1228.505,292.553,-65.810,-176.444,6.701,148.188
C04283=1228.501,292.801,-65.840,-176.442,6.704,148.188
C04284=1228.497,293.050,-65.869,-176.439,6.706,148.187
C04285=1228.493,293.298,-65.898,-176.437,6.708,148.187
C04286=1228.488,293.546,-65.926,-176.435,6.710,148.187
C04287=1228.484,293.794,-65.955,-176.432,6.713,148.187
C04288=1228.480,294.043,-65.984,-176.430,6.715,148.187
C04289=1228.475,294.292,-66.013,-176.427,6.717,148.187
C04290=1228.471,294.539,-66.043,-176.425,6.720,148.187
C04291=1228.467,294.788,-66.071,-176.422,6.722,148.187
C04292=1228.463,295.036,-66.100,-176.420,6.725,148.187
C04293=1228.458,295.285,-66.129,-176.418,6.727,148.186
C04294=1228.453,295.532,-66.158,-176.416,6.729,148.186
C04295=1228.449,295.781,-66.187,-176.413,6.732,148.186
C04296=1228.445,296.030,-66.216,-176.411,6.734,148.186
C04297=1228.440,296.278,-66.246,-176.409,6.736,148.186
C04298=1228.436,296.525,-66.275,-176.406,6.738,148.186
C04299=1228.432,296.773,-66.304,-176.404,6.741,148.186
C04300=1228.428,297.022,-66.332,-176.401,6.743,148.186
C04301=1228.424,297.271,-66.362,-176.399,6.746,148.186
C04302=1228.419,297.519,-66.391,-176.397,6.748,148.186
C04303=1228.414,297.767,-66.420,-176.394,6.751,148.186
C04304=1228.410,298.015,-66.449,-176.392,6.753,148.186
C04305=1228.406,298.264,-66.478,-176.390,6.755,148.185
C04306=1228.402,298.512,-66.508,-176.387,6.758,148.185
C04307=1228.398,298.760,-66.537,-176.385,6.760,148.185
C04308=1228.393,299.008,-66.566,-176.383,6.762,148.185
C04309=1228.388,299.256,-66.595,-176.381,6.765,148.185
C04310=1228.384,299.505,-66.625,-176.378,6.768,148.185
C04311=1228.380,299.753,-66.654,-176.375,6.770,148.185
C04312=1228.376,300.001,-66.684,-176.373,6.772,148.185
C04313=1228.372,300.250,-66.713,-176.371,6.774,148.185
C04314=1228.367,300.498,-66.742,-176.369,6.777,148.185
C04315=1228.362,300.746,-66.771,-176.366,6.779,148.185
C04316=1228.358,300.994,-66.800,-176.364,6.782,148.185
C04317=1228.354,301.243,-66.830,-176.362,6.785,148.185
C04318=1228.350,301.491,-66.859,-176.359,6.787,148.184
C04319=1228.346,301.739,-66.889,-176.357,6.789,148.184
C04320=1228.341,301.987,-66.918,-176.355,6.791,148.184
C04321=1228.337,302.236,-66.948,-176.352,6.794,148.184
C04322=1228.332,302.483,-66.977,-176.350,6.796,148.184
C04323=1228.328,302.731,-67.006,-176.348,6.798,148.184
C04324=1228.324,302.980,-67.036,-176.345,6.802,148.184
C04325=1228.320,303.228,-67.065,-176.343,6.804,148.184
C04326=1228.316,303.476,-67.094,-176.341,6.806,148.184
C04327=1228.311,303.725,-67.125,-176.339,6.808,148.184
C04328=1228.307,303.973,-67.154,-176.336,6.811,148.184
C04329=1228.302,304.221,-67.183,-176.334,6.813,148.184
C04330=1228.298,304.470,-67.213,-176.332,6.815,148.184
C04331=1228.294,304.718,-67.242,-176.329,6.818,148.184
C04332=1228.290,304.966,-67.272,-176.327,6.821,148.183
C04333=1228.285,305.214,-67.301,-176.325,6.823,148.183
C04334=1228.280,305.462,-67.331,-176.323,6.825,148.183
C04335=1228.276,305.710,-67.361,-176.320,6.828,148.183
C04336=1228.272,305.958,-67.391,-176.318,6.830,148.183
C04337=1228.268,306.206,-67.420,-176.316,6.833,148.183
C04338=1228.264,306.455,-67.449,-176.313,6.836,148.183
C04339=1228.260,306.703,-67.479,-176.311,6.838,148.183
C04340=1228.255,306.952,-67.509,-176.309,6.840,148.183
C04341=1228.251,307.199,-67.539,-176.307,6.842,148.183
C04342=1228.247,307.448,-67.569,-176.304,6.845,148.183
C04343=1228.242,307.696,-67.598,-176.302,6.848,148.183
C04344=1228.238,307.944,-67.628,-176.300,6.850,148.183
C04345=1228.233,308.193,-67.658,-176.297,6.853,148.183
C04346=1228.229,308.440,-67.688,-176.295,6.855,148.183
C04347=1228.225,308.689,-67.717,-176.293,6.857,148.183
C04348=1228.220,308.937,-67.747,-176.290,6.860,148.183
C04349=1228.216,309.185,-67.777,-176.288,6.863,148.183
C04350=1228.212,309.433,-67.807,-176.286,6.865,148.183
C04351=1228.208,309.681,-67.836,-176.284,6.867,148.183
C04352=1228.203,309.930,-67.866,-176.282,6.870,148.183
C04353=1228.199,310.178,-67.897,-176.279,6.872,148.183
C04354=1228.195,310.426,-67.926,-176.277,6.875,148.183
C04355=1228.190,310.674,-67.956,-176.275,6.878,148.183
C04356=1228.186,310.922,-67.986,-176.273,6.880,148.183
C04357=1228.182,311.170,-68.016,-176.270,6.882,148.183
C04358=1228.177,311.419,-68.046,-176.268,6.885,148.183
C04359=1228.173,311.667,-68.076,-176.266,6.887,148.182
C04360=1228.169,311.915,-68.105,-176.264,6.890,148.182
C04361=1228.165,312.163,-68.136,-176.261,6.893,148.182
C04362=1228.160,312.411,-68.166,-176.259,6.895,148.182
C04363=1228.156,312.659,-68.195,-176.257,6.897,148.182
C04364=1228.152,312.907,-68.226,-176.255,6.899,148.182
C04365=1228.148,313.156,-68.256,-176.252,6.902,148.182
C04366=1228.144,313.404,-68.286,-176.250,6.905,148.182
C04367=1228.139,313.652,-68.316,-176.248,6.907,148.182
C04368=1228.135,313.900,-68.346,-176.246,6.910,148.182
C04369=1228.130,314.149,-68.376,-176.243,6.912,148.182
C04370=1228.127,314.396,-68.406,-176.241,6.915,148.182
C04371=1228.122,314.645,-68.436,-176.239,6.918,148.182
C04372=1228.118,314.893,-68.466,-176.237,6.920,148.182
C04373=1228.113,315.169,-68.499,-176.234,6.923,148.182
C04374=1228.109,315.444,-68.534,-176.232,6.925,148.182
C04375=1228.103,315.720,-68.567,-176.229,6.928,148.182
C04376=1228.099,315.996,-68.601,-176.227,6.931,148.182
C04377=1228.094,316.244,-68.631,-176.224,6.934,148.182
C04378=1228.090,316.492,-68.661,-176.222,6.936,148.182
C04379=1228.086,316.739,-68.691,-176.220,6.939,148.182
C04380=1228.082,316.989,-68.721,-176.218,6.941,148.182
C04381=1228.078,317.236,-68.751,-176.216,6.944,148.182
C04382=1228.073,317.484,-68.782,-176.213,6.947,148.182
C04383=1228.069,317.733,-68.812,-176.211,6.949,148.182
C04384=1228.065,317.981,-68.842,-176.210,6.951,148.182
C04385=1228.060,318.229,-68.873,-176.207,6.954,148.182
C04386=1228.056,318.478,-68.903,-176.205,6.957,148.182
C04387=1228.052,318.725,-68.934,-176.203,6.959,148.182
C04388=1228.048,318.973,-68.964,-176.201,6.961,148.182
C04389=1228.043,319.222,-68.994,-176.198,6.964,148.182
C04390=1228.039,319.469,-69.024,-176.196,6.967,148.182
C04391=1228.035,319.717,-69.055,-176.194,6.969,148.182
C04392=1228.031,319.966,-69.085,-176.192,6.972,148.182
C04393=1228.027,320.214,-69.116,-176.190,6.974,148.182
C04394=1228.022,320.462,-69.146,-176.188,6.977,148.182
C04395=1228.018,320.710,-69.176,-176.185,6.980,148.182
C04396=1228.013,320.958,-69.207,-176.183,6.982,148.182
C04397=1228.010,321.206,-69.238,-176.181,6.984,148.182
C04398=1228.005,321.454,-69.269,-176.179,6.988,148.183
C04399=1228.000,321.703,-69.299,-176.177,6.990,148.183
C04400=1227.997,321.950,-69.329,-176.175,6.992,148.183
C04401=1227.993,322.199,-69.360,-176.172,6.995,148.183
C04402=1227.988,322.447,-69.391,-176.170,6.998,148.183
C04403=1227.984,322.695,-69.421,-176.168,7.000,148.183
C04404=1227.979,322.943,-69.452,-176.166,7.003,148.183
C04405=1227.975,323.191,-69.483,-176.164,7.005,148.183
C04406=1227.972,323.439,-69.513,-176.162,7.008,148.183
C04407=1227.967,323.687,-69.544,-176.159,7.011,148.183
C04408=1227.962,323.935,-69.574,-176.158,7.013,148.183
C04409=1227.959,324.183,-69.605,-176.156,7.015,148.183
C04410=1227.954,324.432,-69.635,-176.153,7.018,148.183
C04411=1227.950,324.680,-69.666,-176.151,7.021,148.183
C04412=1227.945,324.928,-69.697,-176.149,7.023,148.183
C04413=1227.942,325.176,-69.727,-176.147,7.026,148.183
C04414=1227.937,325.424,-69.758,-176.145,7.029,148.183
C04415=1227.933,325.671,-69.789,-176.143,7.031,148.183
C04416=1227.929,325.920,-69.820,-176.141,7.033,148.183
C04417=1227.925,326.168,-69.851,-176.138,7.037,148.183
C04418=1227.920,326.416,-69.881,-176.136,7.039,148.183
C04419=1227.916,326.664,-69.912,-176.134,7.041,148.183
C04420=1227.912,326.912,-69.943,-176.132,7.045,148.184
C04421=1227.908,327.160,-69.973,-176.130,7.047,148.183
C04422=1227.903,327.408,-70.004,-176.128,7.049,148.184
C04423=1227.899,327.656,-70.035,-176.126,7.052,148.184
C04424=1227.894,327.904,-70.066,-176.124,7.055,148.184
C04425=1227.890,328.152,-70.097,-176.122,7.057,148.184
C04426=1227.887,328.400,-70.128,-176.119,7.060,148.184
C04427=1227.882,328.648,-70.159,-176.118,7.063,148.184
C04428=1227.878,328.897,-70.190,-176.116,7.065,148.184
C04429=1227.874,329.145,-70.221,-176.113,7.068,148.184
C04430=1227.869,329.393,-70.252,-176.111,7.071,148.184
C04431=1227.865,329.641,-70.283,-176.109,7.073,148.184
C04432=1227.861,329.888,-70.314,-176.108,7.075,148.184
C04433=1227.857,330.136,-70.344,-176.105,7.078,148.184
C04434=1227.853,330.385,-70.375,-176.103,7.081,148.184
C04435=1227.848,330.633,-70.406,-176.101,7.083,148.184
C04436=1227.844,330.880,-70.438,-176.099,7.086,148.185
C04437=1227.840,331.129,-70.469,-176.097,7.089,148.185
C04438=1227.835,331.377,-70.500,-176.095,7.091,148.185
C04439=1227.831,331.625,-70.531,-176.093,7.094,148.185
C04440=1227.827,331.873,-70.562,-176.091,7.097,148.185
C04441=1227.822,332.121,-70.593,-176.089,7.099,148.185
C04442=1227.818,332.369,-70.624,-176.087,7.102,148.185
C04443=1227.814,332.617,-70.656,-176.085,7.105,148.185
C04444=1227.811,332.865,-70.686,-176.083,7.107,148.185
C04445=1227.806,333.113,-70.717,-176.080,7.110,148.185
C04446=1227.802,333.360,-70.748,-176.079,7.113,148.185
C04447=1227.798,333.609,-70.779,-176.077,7.115,148.185
C04448=1227.793,333.857,-70.810,-176.075,7.117,148.186
C04449=1227.790,334.105,-70.842,-176.072,7.121,148.186
C04450=1227.785,334.353,-70.873,-176.071,7.123,148.186
C04451=1227.781,334.601,-70.905,-176.069,7.126,148.186
C04452=1227.777,334.849,-70.935,-176.067,7.129,148.186
C04453=1227.772,335.096,-70.967,-176.065,7.131,148.186
C04454=1227.768,335.345,-70.998,-176.063,7.133,148.186
C04455=1227.764,335.592,-71.030,-176.061,7.137,148.186
C04456=1227.760,335.841,-71.061,-176.059,7.139,148.187
C04457=1227.755,336.089,-71.092,-176.057,7.142,148.186
C04458=1227.751,336.337,-71.124,-176.055,7.145,148.187
C04459=1227.746,336.585,-71.155,-176.053,7.147,148.187
C04460=1227.743,336.833,-71.186,-176.051,7.150,148.187
C04461=1227.738,337.081,-71.218,-176.049,7.152,148.187
C04462=1227.734,337.329,-71.249,-176.047,7.155,148.187
C04463=1227.730,337.577,-71.281,-176.045,7.158,148.187
C04464=1227.726,337.825,-71.312,-176.043,7.160,148.187
C04465=1227.722,338.073,-71.343,-176.041,7.163,148.187
C04466=1227.718,338.321,-71.374,-176.039,7.166,148.188
C04467=1227.713,338.569,-71.406,-176.038,7.168,148.188
C04468=1227.710,338.817,-71.438,-176.035,7.172,148.188
C04469=1227.704,339.065,-71.469,-176.033,7.174,148.188
C04470=1227.701,339.313,-71.501,-176.032,7.177,148.188
C04471=1227.696,339.561,-71.532,-176.030,7.179,148.188
C04472=1227.692,339.809,-71.563,-176.027,7.182,148.188
C04473=1227.688,340.056,-71.595,-176.026,7.185,148.189
C04474=1227.684,340.305,-71.626,-176.024,7.187,148.189
C04475=1227.680,340.552,-71.658,-176.021,7.190,148.189
C04476=1227.675,340.801,-71.690,-176.020,7.193,148.189
C04477=1227.671,341.079,-71.725,-176.018,7.196,148.189
C04478=1227.666,341.356,-71.760,-176.016,7.198,148.189
C04479=1227.661,341.633,-71.796,-176.013,7.202,148.189
C04480=1227.657,341.911,-71.831,-176.011,7.205,148.190
C04481=1227.652,342.160,-71.863,-176.010,7.208,148.190
C04482=1227.648,342.407,-71.895,-176.008,7.210,148.190
C04483=1227.644,342.655,-71.926,-176.006,7.212,148.190
C04484=1227.640,342.903,-71.957,-176.004,7.216,148.190
C04485=1227.635,343.151,-71.990,-176.002,7.218,148.190
C04486=1227.631,343.399,-72.021,-176.000,7.221,148.190
C04487=1227.627,343.647,-72.053,-175.998,7.224,148.190
C04488=1227.623,343.895,-72.085,-175.996,7.226,148.191
C04489=1227.618,344.143,-72.116,-175.995,7.229,148.191
C04490=1227.614,344.391,-72.148,-175.993,7.232,148.191
C04491=1227.610,344.638,-72.179,-175.991,7.235,148.191
C04492=1227.606,344.887,-72.212,-175.989,7.237,148.191
C04493=1227.602,345.135,-72.244,-175.988,7.240,148.192
C04494=1227.598,345.382,-72.275,-175.985,7.242,148.192
C04495=1227.594,345.630,-72.307,-175.983,7.246,148.192
C04496=1227.589,345.878,-72.339,-175.982,7.248,148.192
C04497=1227.585,346.126,-72.370,-175.980,7.251,148.192
C04498=1227.581,346.375,-72.402,-175.978,7.253,148.192
C04499=1227.576,346.622,-72.434,-175.976,7.256,148.193
C04500=1227.572,346.870,-72.466,-175.975,7.259,148.193
C04501=1227.569,347.118,-72.498,-175.973,7.262,148.193
C04502=1227.564,347.366,-72.530,-175.971,7.264,148.193
C04503=1227.560,347.614,-72.562,-175.969,7.267,148.193
C04504=1227.555,347.862,-72.594,-175.967,7.270,148.193
C04505=1227.551,348.110,-72.626,-175.965,7.272,148.194
C04506=1227.547,348.358,-72.658,-175.964,7.275,148.194
C04507=1227.543,348.606,-72.690,-175.962,7.278,148.194
C04508=1227.539,348.853,-72.721,-175.960,7.281,148.194
C04509=1227.534,349.102,-72.754,-175.958,7.283,148.194
C04510=1227.531,349.350,-72.786,-175.957,7.286,148.194
C04511=1227.526,349.597,-72.817,-175.955,7.289,148.195
C04512=1227.522,349.845,-72.850,-175.953,7.292,148.195
C04513=1227.518,350.093,-72.882,-175.951,7.294,148.195
C04514=1227.513,350.340,-72.914,-175.950,7.297,148.195
C04515=1227.510,350.589,-72.946,-175.947,7.300,148.196
C04516=1227.505,350.837,-72.979,-175.946,7.303,148.196
C04517=1227.501,351.084,-73.010,-175.944,7.305,148.196
C04518=1227.497,351.332,-73.042,-175.943,7.308,148.196
C04519=1227.493,351.581,-73.074,-175.940,7.311,148.196
C04520=1227.489,351.829,-73.106,-175.939,7.313,148.196
C04521=1227.484,352.076,-73.139,-175.937,7.316,148.197
C04522=1227.481,352.324,-73.171,-175.936,7.319,148.197
C04523=1227.476,352.572,-73.203,-175.934,7.321,148.197
C04524=1227.472,352.820,-73.235,-175.932,7.325,148.197
C04525=1227.467,353.068,-73.267,-175.931,7.327,148.198
C04526=1227.464,353.315,-73.300,-175.929,7.330,148.198
C04527=1227.460,353.563,-73.332,-175.927,7.332,148.198
C04528=1227.455,353.811,-73.364,-175.925,7.336,148.198
C04529=1227.451,354.059,-73.396,-175.923,7.338,148.198
C04530=1227.447,354.307,-73.429,-175.922,7.341,148.199
C04531=1227.443,354.555,-73.461,-175.920,7.343,148.199
C04532=1227.439,354.803,-73.494,-175.919,7.346,148.199
C04533=1227.434,355.051,-73.525,-175.917,7.349,148.199
C04534=1227.430,355.298,-73.558,-175.915,7.352,148.200
C04535=1227.426,355.546,-73.590,-175.914,7.354,148.200
C04536=1227.422,355.795,-73.622,-175.912,7.357,148.200
C04537=1227.418,356.041,-73.655,-175.910,7.360,148.200
C04538=1227.414,356.290,-73.687,-175.909,7.363,148.201
C04539=1227.409,356.538,-73.720,-175.907,7.366,148.201
C04540=1227.406,356.786,-73.752,-175.905,7.368,148.201
C04541=1227.401,357.034,-73.785,-175.904,7.371,148.201
C04542=1227.397,357.281,-73.816,-175.902,7.373,148.201
C04543=1227.393,357.529,-73.849,-175.901,7.376,148.202
C04544=1227.388,357.777,-73.882,-175.899,7.380,148.202
C04545=1227.385,358.025,-73.914,-175.897,7.382,148.202
C04546=1227.380,358.273,-73.947,-175.896,7.385,148.202
C04547=1227.376,358.520,-73.979,-175.894,7.387,148.203
C04548=1227.372,358.768,-74.011,-175.893,7.390,148.203
C04549=1227.368,359.017,-74.044,-175.891,7.392,148.203
C04550=1227.363,359.264,-74.077,-175.889,7.396,148.203
C04551=1227.360,359.512,-74.109,-175.888,7.399,148.204
C04552=1227.356,359.760,-74.142,-175.886,7.401,148.204
C04553=1227.351,360.008,-74.174,-175.885,7.404,148.204
C04554=1227.347,360.255,-74.206,-175.883,7.407,148.205
C04555=1227.343,360.503,-74.239,-175.882,7.409,148.205
C04556=1227.339,360.751,-74.272,-175.880,7.412,148.205
C04557=1227.335,360.999,-74.304,-175.878,7.415,148.205
C04558=1227.331,361.247,-74.337,-175.877,7.418,148.206
C04559=1227.326,361.495,-74.370,-175.875,7.420,148.206
C04560=1227.322,361.743,-74.403,-175.874,7.423,148.206
C04561=1227.318,361.990,-74.435,-175.872,7.426,148.206
C04562=1227.314,362.238,-74.467,-175.871,7.428,148.206
C04563=1227.310,362.486,-74.500,-175.870,7.431,148.207
C04564=1227.305,362.734,-74.533,-175.867,7.434,148.207
C04565=1227.302,362.982,-74.565,-175.866,7.437,148.208
C04566=1227.298,363.229,-74.599,-175.865,7.440,148.208
C04567=1227.293,363.478,-74.631,-175.863,7.443,148.208
C04568=1227.289,363.725,-74.664,-175.862,7.445,148.208
C04569=1227.286,363.973,-74.697,-175.860,7.448,148.208
C04570=1227.281,364.220,-74.729,-175.859,7.450,148.209
C04571=1227.276,364.468,-74.762,-175.857,7.453,148.209
C04572=1227.272,364.716,-74.795,-175.856,7.456,148.209
C04573=1227.268,364.964,-74.828,-175.854,7.459,148.210
C04574=1227.264,365.212,-74.860,-175.853,7.462,148.210
C04575=1227.260,365.459,-74.893,-175.851,7.465,148.210
C04576=1227.256,365.708,-74.926,-175.850,7.467,148.211
C04577=1227.252,365.956,-74.959,-175.848,7.470,148.211
C04578=1227.248,366.203,-74.992,-175.847,7.473,148.211
C04579=1227.244,366.451,-75.025,-175.846,7.475,148.211
C04580=1227.240,366.699,-75.057,-175.844,7.478,148.212
C04581=1227.235,366.979,-75.095,-175.842,7.481,148.212
C04582=1227.230,367.257,-75.132,-175.841,7.484,148.212
C04583=1227.225,367.538,-75.169,-175.840,7.487,148.213
C04584=1227.220,367.817,-75.206,-175.838,7.490,148.213
C04585=1227.217,368.065,-75.239,-175.837,7.493,148.214
C04586=1227.213,368.312,-75.272,-175.835,7.496,148.214
C04587=1227.208,368.561,-75.304,-175.834,7.499,148.214
C04588=1227.204,368.808,-75.337,-175.833,7.501,148.215
C04589=1227.200,369.056,-75.371,-175.831,7.504,148.215
C04590=1227.196,369.304,-75.404,-175.830,7.507,148.215
C04591=1227.192,369.552,-75.437,-175.828,7.509,148.215
C04592=1227.188,369.799,-75.470,-175.827,7.512,148.216
C04593=1227.183,370.048,-75.502,-175.826,7.515,148.216
C04594=1227.179,370.295,-75.536,-175.824,7.517,148.216
C04595=1227.175,370.543,-75.569,-175.823,7.520,148.217
C04596=1227.171,370.791,-75.602,-175.822,7.523,148.217
C04597=1227.167,371.039,-75.635,-175.820,7.526,148.217
C04598=1227.163,371.286,-75.668,-175.819,7.528,148.218
C04599=1227.159,371.534,-75.701,-175.818,7.531,148.218
C04600=1227.155,371.782,-75.734,-175.816,7.534,148.218
C04601=1227.151,372.029,-75.767,-175.815,7.537,148.219
C04602=1227.147,372.277,-75.800,-175.814,7.539,148.219
C04603=1227.143,372.525,-75.833,-175.813,7.542,148.219
C04604=1227.139,372.772,-75.867,-175.811,7.545,148.220
C04605=1227.134,373.020,-75.900,-175.810,7.548,148.220
C04606=1227.130,373.268,-75.933,-175.809,7.550,148.220
C04607=1227.126,373.516,-75.966,-175.808,7.553,148.221
C04608=1227.122,373.763,-75.999,-175.806,7.556,148.221
C04609=1227.118,374.011,-76.032,-175.805,7.558,148.221
C04610=1227.114,374.259,-76.066,-175.804,7.561,148.222
C04611=1227.110,374.507,-76.099,-175.803,7.563,148.222
C04612=1227.105,374.754,-76.132,-175.801,7.566,148.222
C04613=1227.101,375.002,-76.166,-175.800,7.569,148.223
C04614=1227.096,375.250,-76.199,-175.799,7.572,148.223
C04615=1227.092,375.498,-76.232,-175.798,7.574,148.224
C04616=1227.089,375.746,-76.265,-175.797,7.577,148.224
C04617=1227.085,375.994,-76.299,-175.796,7.580,148.224
C04618=1227.080,376.242,-76.332,-175.794,7.583,148.225
C04619=1227.076,376.489,-76.365,-175.793,7.585,148.225
C04620=1227.072,376.737,-76.398,-175.792,7.587,148.225
C04621=1227.068,376.984,-76.432,-175.791,7.590,148.226
C04622=1227.064,377.232,-76.465,-175.790,7.593,148.226
C04623=1227.060,377.480,-76.498,-175.789,7.596,148.226
C04624=1227.056,377.727,-76.531,-175.788,7.599,148.227
C04625=1227.052,377.975,-76.565,-175.786,7.601,148.227
C04626=1227.047,378.223,-76.598,-175.785,7.603,148.227
C04627=1227.043,378.471,-76.631,-175.784,7.606,148.228
C04628=1227.040,378.719,-76.666,-175.783,7.609,148.228
C04629=1227.035,378.966,-76.699,-175.782,7.612,148.229
C04630=1227.031,379.214,-76.732,-175.781,7.615,148.229
C04631=1227.027,379.462,-76.765,-175.779,7.617,148.229
C04632=1227.023,379.710,-76.798,-175.779,7.619,148.230
C04633=1227.018,379.957,-76.833,-175.778,7.622,148.230
C04634=1227.014,380.205,-76.866,-175.776,7.625,148.231
C04635=1227.010,380.453,-76.899,-175.775,7.628,148.231
C04636=1227.006,380.700,-76.932,-175.774,7.631,148.231
C04637=1227.003,380.948,-76.966,-175.774,7.633,148.232
C04638=1226.999,381.196,-77.000,-175.772,7.635,148.232
C04639=1226.994,381.444,-77.033,-175.771,7.638,148.232
C04640=1226.990,381.692,-77.067,-175.770,7.641,148.233
C04641=1226.986,381.939,-77.100,-175.769,7.643,148.233
C04642=1226.982,382.186,-77.134,-175.768,7.646,148.234
C04643=1226.978,382.434,-77.167,-175.767,7.649,148.234
C04644=1226.974,382.682,-77.202,-175.766,7.652,148.234
C04645=1226.969,382.930,-77.235,-175.765,7.654,148.235
C04646=1226.965,383.178,-77.268,-175.764,7.656,148.235
C04647=1226.961,383.425,-77.302,-175.763,7.659,148.236
C04648=1226.957,383.673,-77.335,-175.762,7.662,148.236
C04649=1226.952,383.921,-77.369,-175.761,7.664,148.236
C04650=1226.949,384.168,-77.403,-175.760,7.667,148.237
C04651=1226.945,384.416,-77.436,-175.759,7.670,148.237
C04652=1226.941,384.664,-77.469,-175.758,7.672,148.237
C04653=1226.936,384.911,-77.504,-175.757,7.674,148.238
C04654=1226.932,385.159,-77.537,-175.756,7.677,148.238
C04655=1226.928,385.407,-77.570,-175.755,7.680,148.239
C04656=1226.924,385.654,-77.604,-175.754,7.682,148.239
C04657=1226.920,385.903,-77.638,-175.753,7.685,148.239
C04658=1226.916,386.150,-77.672,-175.752,7.688,148.240
C04659=1226.912,386.397,-77.705,-175.751,7.690,148.240
C04660=1226.907,386.645,-77.739,-175.750,7.692,148.240
C04661=1226.903,386.893,-77.773,-175.749,7.696,148.241
C04662=1226.900,387.141,-77.806,-175.748,7.698,148.241
C04663=1226.896,387.388,-77.840,-175.747,7.700,148.242
C04664=1226.891,387.636,-77.874,-175.746,7.703,148.242
C04665=1226.887,387.883,-77.908,-175.746,7.705,148.243
C04666=1226.883,388.131,-77.941,-175.744,7.708,148.243
C04667=1226.879,388.379,-77.976,-175.743,7.711,148.243
C04668=1226.875,388.627,-78.009,-175.743,7.713,148.244
C04669=1226.871,388.874,-78.043,-175.741,7.716,148.244
C04670=1226.866,389.122,-78.076,-175.741,7.718,148.245
C04671=1226.863,389.370,-78.111,-175.740,7.721,148.245
C04672=1226.859,389.618,-78.144,-175.739,7.724,148.245
C04673=1226.854,389.865,-78.178,-175.738,7.726,148.246
C04674=1226.850,390.113,-78.211,-175.737,7.728,148.246
C04675=1226.846,390.360,-78.245,-175.736,7.730,148.247
C04676=1226.842,390.609,-78.279,-175.736,7.733,148.247
C04677=1226.838,390.856,-78.313,-175.735,7.736,148.248
C04678=1226.834,391.103,-78.347,-175.734,7.738,148.248
C04679=1226.830,391.351,-78.381,-175.733,7.741,148.248
C04680=1226.826,391.599,-78.415,-175.732,7.743,148.249
C04681=1226.821,391.847,-78.449,-175.731,7.746,148.249
C04682=1226.818,392.094,-78.483,-175.731,7.748,148.250
C04683=1226.814,392.341,-78.517,-175.730,7.751,148.250
C04684=1226.810,392.590,-78.551,-175.729,7.753,148.250
C04685=1226.805,392.870,-78.589,-175.728,7.756,148.251
C04686=1226.800,393.152,-78.627,-175.727,7.759,148.251
C04687=1226.796,393.433,-78.666,-175.726,7.762,148.252
C04688=1226.791,393.716,-78.705,-175.725,7.765,148.252
C04689=1226.787,393.963,-78.739,-175.725,7.767,148.253
C04690=1226.783,394.210,-78.773,-175.723,7.770,148.253
C04691=1226.778,394.458,-78.806,-175.723,7.772,148.253
C04692=1226.775,394.706,-78.841,-175.722,7.774,148.254
C04693=1226.771,394.953,-78.875,-175.721,7.777,148.254
C04694=1226.767,395.201,-78.908,-175.720,7.780,148.255
C04695=1226.763,395.449,-78.943,-175.720,7.782,148.255
C04696=1226.759,395.696,-78.977,-175.718,7.784,148.255
C04697=1226.754,395.944,-79.011,-175.718,7.787,148.256
C04698=1226.750,396.191,-79.045,-175.717,7.789,148.256
C04699=1226.746,396.439,-79.079,-175.716,7.791,148.257
C04700=1226.742,396.687,-79.113,-175.715,7.794,148.257
C04701=1226.737,396.935,-79.147,-175.715,7.797,148.258
C04702=1226.734,397.182,-79.181,-175.714,7.798,148.258
C04703=1226.730,397.430,-79.216,-175.713,7.801,148.258
C04704=1226.726,397.677,-79.250,-175.713,7.803,148.259
C04705=1226.721,397.926,-79.284,-175.712,7.806,148.259
C04706=1226.718,398.173,-79.318,-175.711,7.808,148.260
C04707=1226.713,398.420,-79.352,-175.710,7.811,148.260
C04708=1226.710,398.668,-79.386,-175.710,7.813,148.261
C04709=1226.705,398.916,-79.420,-175.709,7.815,148.261
C04710=1226.701,399.163,-79.454,-175.708,7.818,148.261
C04711=1226.697,399.411,-79.489,-175.707,7.820,148.262
C04712=1226.693,399.658,-79.523,-175.707,7.823,148.262
C04713=1226.689,399.906,-79.557,-175.706,7.825,148.263
C04714=1226.685,400.154,-79.591,-175.706,7.827,148.263
C04715=1226.681,400.402,-79.625,-175.704,7.830,148.263
C04716=1226.677,400.649,-79.659,-175.704,7.832,148.264
C04717=1226.673,400.897,-79.694,-175.704,7.834,148.264
C04718=1226.669,401.144,-79.728,-175.702,7.837,148.265
C04719=1226.664,401.391,-79.762,-175.702,7.840,148.265
C04720=1226.661,401.639,-79.796,-175.701,7.842,148.266
C04721=1226.656,401.887,-79.830,-175.700,7.844,148.266
C04722=1226.652,402.135,-79.865,-175.700,7.847,148.267
C04723=1226.649,402.383,-79.899,-175.699,7.849,148.267
C04724=1226.644,402.630,-79.933,-175.698,7.851,148.267
C04725=1226.640,402.877,-79.967,-175.698,7.853,148.268
C04726=1226.636,403.125,-80.002,-175.698,7.856,148.268
C04727=1226.632,403.372,-80.036,-175.696,7.858,148.269
C04728=1226.628,403.620,-80.070,-175.696,7.860,148.269
C04729=1226.624,403.868,-80.105,-175.696,7.863,148.269
C04730=1226.620,404.116,-80.138,-175.694,7.866,148.270
C04731=1226.616,404.364,-80.173,-175.694,7.867,148.270
C04732=1226.612,404.611,-80.207,-175.694,7.870,148.271
C04733=1226.607,404.858,-80.242,-175.692,7.873,148.271
C04734=1226.603,405.106,-80.276,-175.692,7.875,148.271
C04735=1226.599,405.353,-80.310,-175.692,7.877,148.272
C04736=1226.595,405.601,-80.345,-175.691,7.879,148.272
C04737=1226.592,405.849,-80.379,-175.690,7.882,148.273
C04738=1226.587,406.096,-80.413,-175.690,7.884,148.273
C04739=1226.583,406.344,-80.448,-175.689,7.886,148.274
C04740=1226.579,406.591,-80.482,-175.688,7.888,148.274
C04741=1226.575,406.839,-80.517,-175.687,7.891,148.274
C04742=1226.571,407.087,-80.551,-175.687,7.893,148.275
C04743=1226.567,407.334,-80.585,-175.686,7.895,148.275
C04744=1226.563,407.582,-80.620,-175.686,7.897,148.276
C04745=1226.558,407.829,-80.655,-175.685,7.900,148.276
C04746=1226.555,408.077,-80.689,-175.684,7.902,148.277
C04747=1226.551,408.325,-80.723,-175.684,7.904,148.277
C04748=1226.546,408.572,-80.758,-175.684,7.906,148.277
C04749=1226.543,408.820,-80.792,-175.682,7.909,148.278
C04750=1226.538,409.067,-80.826,-175.682,7.911,148.278
C04751=1226.534,409.315,-80.861,-175.682,7.913,148.279
C04752=1226.530,409.563,-80.895,-175.681,7.915,148.279
C04753=1226.526,409.810,-80.930,-175.680,7.917,148.279
C04754=1226.522,410.058,-80.965,-175.680,7.920,148.280
C04755=1226.518,410.305,-80.999,-175.679,7.922,148.280
C04756=1226.514,410.553,-81.034,-175.678,7.924,148.281
C04757=1226.510,410.800,-81.068,-175.678,7.927,148.281
C04758=1226.507,411.048,-81.103,-175.677,7.929,148.282
C04759=1226.502,411.295,-81.137,-175.677,7.931,148.282
C04760=1226.498,411.544,-81.172,-175.676,7.934,148.283
C04761=1226.494,411.791,-81.206,-175.675,7.936,148.283
C04762=1226.490,412.038,-81.240,-175.675,7.938,148.283
C04763=1226.486,412.286,-81.275,-175.675,7.940,148.284
C04764=1226.481,412.533,-81.310,-175.674,7.942,148.284
C04765=1226.478,412.781,-81.344,-175.673,7.944,148.284
C04766=1226.474,413.028,-81.379,-175.673,7.947,148.285
C04767=1226.470,413.276,-81.414,-175.672,7.949,148.285
C04768=1226.465,413.524,-81.448,-175.671,7.951,148.286
C04769=1226.462,413.772,-81.482,-175.671,7.953,148.286
C04770=1226.457,414.019,-81.517,-175.671,7.955,148.287
C04771=1226.453,414.266,-81.552,-175.670,7.957,148.287
C04772=1226.450,414.514,-81.586,-175.669,7.959,148.287
C04773=1226.445,414.761,-81.621,-175.669,7.961,148.288
C04774=1226.441,415.009,-81.656,-175.668,7.964,148.288
C04775=1226.437,415.257,-81.690,-175.667,7.966,148.289
C04776=1226.433,415.504,-81.726,-175.667,7.968,148.289
C04777=1226.426,415.901,-81.781,-175.666,7.972,148.290
C04778=1226.420,416.298,-81.836,-175.665,7.976,148.290
C04779=1226.414,416.695,-81.891,-175.664,7.979,148.291
C04780=1226.409,417.093,-81.947,-175.664,7.982,148.292
C04781=1225.987,417.092,-81.981,-175.667,7.992,148.295
C04782=1225.992,416.693,-81.925,-175.667,7.989,148.295
C04783=1225.998,416.292,-81.869,-175.669,7.985,148.294
C04784=1226.005,415.893,-81.812,-175.669,7.982,148.293
C04785=1226.011,415.493,-81.757,-175.670,7.979,148.293
C04786=1226.016,415.246,-81.722,-175.671,7.977,148.292
C04787=1226.019,414.998,-81.688,-175.671,7.974,148.292
C04788=1226.023,414.751,-81.653,-175.672,7.972,148.291
C04789=1226.027,414.503,-81.618,-175.673,7.970,148.291
C04790=1226.032,414.256,-81.583,-175.673,7.968,148.291
C04791=1226.035,414.008,-81.549,-175.674,7.966,148.290
C04792=1226.039,413.761,-81.515,-175.674,7.964,148.290
C04793=1226.043,413.512,-81.480,-175.675,7.962,148.290
C04794=1226.048,413.266,-81.445,-175.675,7.959,148.289
C04795=1226.051,413.019,-81.411,-175.676,7.956,148.289
C04796=1226.055,412.770,-81.376,-175.677,7.955,148.288
C04797=1226.060,412.523,-81.342,-175.677,7.952,148.288
C04798=1226.064,412.275,-81.307,-175.678,7.950,148.287
C04799=1226.068,412.028,-81.273,-175.678,7.948,148.287
C04800=1226.072,411.780,-81.238,-175.679,7.946,148.286
C04801=1226.076,411.533,-81.203,-175.679,7.944,148.286
C04802=1226.080,411.285,-81.168,-175.680,7.941,148.286
C04803=1226.084,411.038,-81.134,-175.681,7.939,148.285
C04804=1226.088,410.790,-81.099,-175.681,7.937,148.285
C04805=1226.092,410.542,-81.065,-175.682,7.935,148.285
C04806=1226.096,410.295,-81.031,-175.682,7.933,148.284
C04807=1226.100,410.047,-80.996,-175.683,7.930,148.284
C04808=1226.105,409.799,-80.962,-175.684,7.928,148.283
C04809=1226.108,409.552,-80.927,-175.684,7.926,148.283
C04810=1226.113,409.304,-80.893,-175.685,7.924,148.282
C04811=1226.117,409.056,-80.858,-175.685,7.922,148.282
C04812=1226.120,408.809,-80.824,-175.686,7.919,148.281
C04813=1226.125,408.562,-80.789,-175.687,7.917,148.281
C04814=1226.129,408.314,-80.754,-175.687,7.915,148.281
C04815=1226.132,408.067,-80.720,-175.687,7.912,148.280
C04816=1226.136,407.819,-80.686,-175.688,7.910,148.280
C04817=1226.141,407.571,-80.651,-175.689,7.908,148.279
C04818=1226.145,407.324,-80.617,-175.689,7.905,148.279
C04819=1226.149,407.076,-80.582,-175.690,7.903,148.279
C04820=1226.153,406.829,-80.548,-175.691,7.901,148.278
C04821=1226.157,406.581,-80.514,-175.691,7.898,148.278
C04822=1226.161,406.334,-80.479,-175.692,7.896,148.277
C04823=1226.166,406.086,-80.445,-175.693,7.894,148.277
C04824=1226.169,405.838,-80.411,-175.693,7.892,148.276
C04825=1226.174,405.591,-80.376,-175.694,7.889,148.276
C04826=1226.177,405.343,-80.342,-175.695,7.887,148.276
C04827=1226.181,405.096,-80.307,-175.695,7.885,148.275
C04828=1226.186,404.848,-80.273,-175.695,7.883,148.275
C04829=1226.189,404.600,-80.239,-175.697,7.880,148.274
C04830=1226.194,404.352,-80.205,-175.697,7.878,148.274
C04831=1226.198,404.104,-80.170,-175.697,7.876,148.273
C04832=1226.202,403.857,-80.136,-175.699,7.873,148.273
C04833=1226.206,403.610,-80.102,-175.699,7.871,148.273
C04834=1226.210,403.362,-80.068,-175.699,7.869,148.272
C04835=1226.214,403.115,-80.033,-175.701,7.866,148.272
C04836=1226.218,402.867,-79.999,-175.701,7.864,148.271
C04837=1226.222,402.619,-79.964,-175.701,7.862,148.271
C04838=1226.227,402.372,-79.930,-175.702,7.860,148.271
C04839=1226.230,402.124,-79.896,-175.703,7.857,148.270
C04840=1226.234,401.877,-79.861,-175.703,7.855,148.270
C04841=1226.238,401.629,-79.828,-175.705,7.852,148.269
C04842=1226.242,401.381,-79.793,-175.705,7.850,148.269
C04843=1226.246,401.134,-79.759,-175.705,7.848,148.268
C04844=1226.251,400.886,-79.725,-175.707,7.845,148.268
C04845=1226.255,400.638,-79.690,-175.707,7.843,148.268
C04846=1226.259,400.391,-79.656,-175.707,7.840,148.267
C04847=1226.263,400.144,-79.622,-175.709,7.838,148.267
C04848=1226.267,399.895,-79.588,-175.709,7.836,148.266
C04849=1226.271,399.648,-79.554,-175.710,7.834,148.266
C04850=1226.275,399.401,-79.520,-175.711,7.831,148.265
C04851=1226.279,399.153,-79.485,-175.711,7.829,148.265
C04852=1226.283,398.905,-79.451,-175.712,7.826,148.265
C04853=1226.288,398.657,-79.417,-175.713,7.824,148.264
C04854=1226.291,398.410,-79.383,-175.713,7.822,148.264
C04855=1226.296,398.162,-79.349,-175.714,7.819,148.263
C04856=1226.299,397.915,-79.315,-175.715,7.817,148.263
C04857=1226.303,397.667,-79.280,-175.716,7.814,148.262
C04858=1226.308,397.419,-79.247,-175.716,7.812,148.262
C04859=1226.312,397.172,-79.212,-175.718,7.809,148.262
C04860=1226.315,396.924,-79.178,-175.718,7.807,148.261
C04861=1226.320,396.677,-79.144,-175.718,7.805,148.261
C04862=1226.324,396.429,-79.110,-175.720,7.802,148.260
C04863=1226.329,396.181,-79.076,-175.720,7.800,148.260
C04864=1226.332,395.934,-79.042,-175.721,7.797,148.259
C04865=1226.337,395.686,-79.008,-175.721,7.795,148.259
C04866=1226.341,395.438,-78.974,-175.723,7.792,148.259
C04867=1226.345,395.190,-78.939,-175.723,7.790,148.258
C04868=1226.348,394.943,-78.905,-175.724,7.787,148.258
C04869=1226.353,394.696,-78.872,-175.725,7.785,148.257
C04870=1226.357,394.448,-78.838,-175.726,7.782,148.257
C04871=1226.360,394.200,-78.804,-175.726,7.780,148.257
C04872=1226.365,393.952,-78.770,-175.728,7.777,148.256
C04873=1226.369,393.705,-78.736,-175.728,7.775,148.256
C04874=1226.373,393.423,-78.698,-175.729,7.772,148.255
C04875=1226.378,393.142,-78.658,-175.730,7.769,148.255
C04876=1226.382,392.860,-78.619,-175.731,7.766,148.254
C04877=1226.388,392.579,-78.582,-175.732,7.763,148.254
C04878=1226.392,392.331,-78.547,-175.733,7.761,148.254
C04879=1226.396,392.083,-78.514,-175.733,7.758,148.253
C04880=1226.399,391.836,-78.480,-175.734,7.756,148.253
C04881=1226.404,391.589,-78.445,-175.735,7.753,148.252
C04882=1226.408,391.340,-78.412,-175.736,7.751,148.252
C04883=1226.412,391.093,-78.377,-175.737,7.749,148.251
C04884=1226.416,390.845,-78.344,-175.738,7.746,148.251
C04885=1226.420,390.598,-78.310,-175.738,7.744,148.251
C04886=1226.424,390.349,-78.276,-175.740,7.741,148.250
C04887=1226.428,390.102,-78.242,-175.740,7.739,148.250
C04888=1226.432,389.855,-78.209,-175.741,7.736,148.249
C04889=1226.437,389.607,-78.175,-175.742,7.734,148.249
C04890=1226.440,389.359,-78.141,-175.743,7.731,148.248
C04891=1226.444,389.111,-78.107,-175.744,7.728,148.248
C04892=1226.449,388.864,-78.073,-175.744,7.726,148.248
C04893=1226.453,388.616,-78.040,-175.746,7.723,148.247
C04894=1226.457,388.369,-78.006,-175.747,7.720,148.247
C04895=1226.461,388.120,-77.972,-175.747,7.718,148.247
C04896=1226.465,387.873,-77.938,-175.749,7.716,148.246
C04897=1226.469,387.626,-77.905,-175.749,7.713,148.246
C04898=1226.474,387.378,-77.870,-175.750,7.710,148.245
C04899=1226.478,387.130,-77.837,-175.751,7.708,148.245
C04900=1226.481,386.883,-77.803,-175.752,7.706,148.244
C04901=1226.486,386.635,-77.769,-175.753,7.703,148.244
C04902=1226.490,386.387,-77.736,-175.754,7.700,148.244
C04903=1226.494,386.140,-77.702,-175.755,7.698,148.243
C04904=1226.499,385.892,-77.668,-175.756,7.695,148.243
C04905=1226.502,385.644,-77.634,-175.757,7.692,148.243
C04906=1226.506,385.396,-77.601,-175.757,7.690,148.242
C04907=1226.510,385.149,-77.567,-175.758,7.687,148.242
C04908=1226.515,384.901,-77.533,-175.760,7.684,148.241
C04909=1226.519,384.653,-77.500,-175.761,7.682,148.241
C04910=1226.522,384.405,-77.466,-175.761,7.680,148.240
C04911=1226.526,384.158,-77.433,-175.763,7.677,148.240
C04912=1226.531,383.910,-77.399,-175.764,7.674,148.240
C04913=1226.535,383.663,-77.365,-175.764,7.672,148.239
C04914=1226.539,383.415,-77.332,-175.766,7.669,148.239
C04915=1226.543,383.167,-77.299,-175.767,7.666,148.239
C04916=1226.547,382.919,-77.264,-175.768,7.664,148.238
C04917=1226.551,382.671,-77.231,-175.769,7.662,148.238
C04918=1226.556,382.424,-77.198,-175.770,7.659,148.237
C04919=1226.559,382.176,-77.164,-175.771,7.656,148.237
C04920=1226.564,381.929,-77.131,-175.772,7.653,148.237
C04921=1226.568,381.681,-77.097,-175.773,7.651,148.236
C04922=1226.572,381.434,-77.063,-175.774,7.648,148.236
C04923=1226.576,381.185,-77.030,-175.775,7.646,148.235
C04924=1226.580,380.937,-76.996,-175.776,7.643,148.235
C04925=1226.584,380.690,-76.963,-175.777,7.640,148.235
C04926=1226.588,380.443,-76.929,-175.778,7.638,148.234
C04927=1226.593,380.195,-76.896,-175.779,7.635,148.234
C04928=1226.597,379.947,-76.862,-175.780,7.632,148.234
C04929=1226.601,379.699,-76.829,-175.781,7.629,148.233
C04930=1226.605,379.452,-76.795,-175.783,7.627,148.233
C04931=1226.609,379.204,-76.762,-175.783,7.625,148.232
C04932=1226.613,378.956,-76.729,-175.784,7.622,148.232
C04933=1226.617,378.708,-76.695,-175.786,7.619,148.232
C04934=1226.622,378.460,-76.662,-175.787,7.616,148.231
C04935=1226.625,378.213,-76.628,-175.788,7.614,148.231
C04936=1226.630,377.965,-76.595,-175.790,7.611,148.231
C04937=1226.634,377.717,-76.562,-175.790,7.609,148.230
C04938=1226.638,377.470,-76.529,-175.791,7.606,148.230
C04939=1226.642,377.222,-76.495,-175.793,7.603,148.229
C04940=1226.646,376.974,-76.462,-175.794,7.600,148.229
C04941=1226.650,376.727,-76.428,-175.795,7.598,148.229
C04942=1226.654,376.478,-76.394,-175.796,7.595,148.228
C04943=1226.658,376.231,-76.361,-175.798,7.592,148.228
C04944=1226.662,375.983,-76.328,-175.799,7.589,148.228
C04945=1226.667,375.735,-76.295,-175.800,7.587,148.227
C04946=1226.671,375.487,-76.262,-175.801,7.585,148.227
C04947=1226.675,375.240,-76.228,-175.802,7.582,148.227
C04948=1226.679,374.992,-76.195,-175.803,7.579,148.226
C04949=1226.683,374.744,-76.162,-175.805,7.576,148.226
C04950=1226.687,374.497,-76.129,-175.806,7.574,148.226
C04951=1226.691,374.249,-76.096,-175.807,7.571,148.225
C04952=1226.696,374.001,-76.063,-175.808,7.568,148.225
C04953=1226.700,373.753,-76.029,-175.809,7.565,148.224
C04954=1226.704,373.506,-75.996,-175.811,7.563,148.224
C04955=1226.708,373.258,-75.963,-175.812,7.560,148.224
C04956=1226.712,373.010,-75.930,-175.813,7.557,148.223
C04957=1226.716,372.762,-75.897,-175.814,7.554,148.223
C04958=1226.720,372.515,-75.864,-175.816,7.552,148.223
C04959=1226.725,372.267,-75.831,-175.817,7.550,148.222
C04960=1226.729,372.019,-75.797,-175.818,7.547,148.222
C04961=1226.733,371.772,-75.764,-175.820,7.544,148.222
C04962=1226.737,371.524,-75.731,-175.821,7.541,148.221
C04963=1226.741,371.276,-75.698,-175.822,7.539,148.221
C04964=1226.745,371.028,-75.665,-175.823,7.536,148.221
C04965=1226.749,370.781,-75.632,-175.825,7.533,148.220
C04966=1226.754,370.533,-75.598,-175.826,7.530,148.220
C04967=1226.758,370.285,-75.565,-175.827,7.528,148.220
C04968=1226.762,370.037,-75.532,-175.829,7.525,148.219
C04969=1226.766,369.790,-75.499,-175.830,7.522,148.219
C04970=1226.770,369.541,-75.467,-175.831,7.519,148.219
C04971=1226.775,369.294,-75.433,-175.833,7.517,148.219
C04972=1226.779,369.046,-75.400,-175.834,7.514,148.218
C04973=1226.782,368.798,-75.368,-175.835,7.512,148.218
C04974=1226.786,368.551,-75.335,-175.837,7.509,148.218
C04975=1226.790,368.303,-75.301,-175.838,7.506,148.217
C04976=1226.794,368.055,-75.268,-175.840,7.503,148.217
C04977=1226.799,367.807,-75.236,-175.841,7.500,148.216
C04978=1226.803,367.527,-75.198,-175.843,7.497,148.216
C04979=1226.808,367.248,-75.161,-175.844,7.494,148.216
C04980=1226.813,366.968,-75.124,-175.846,7.491,148.215
C04981=1226.817,366.688,-75.087,-175.847,7.488,148.215
C04982=1226.821,366.441,-75.054,-175.848,7.485,148.215
C04983=1226.825,366.193,-75.021,-175.851,7.482,148.215
C04984=1226.830,365.945,-74.988,-175.852,7.479,148.214
C04985=1226.834,365.697,-74.955,-175.853,7.477,148.214
C04986=1226.838,365.450,-74.922,-175.855,7.474,148.214
C04987=1226.842,365.202,-74.890,-175.856,7.471,148.213
C04988=1226.846,364.954,-74.857,-175.857,7.468,148.213
C04989=1226.850,364.706,-74.824,-175.859,7.466,148.213
C04990=1226.855,364.459,-74.791,-175.860,7.463,148.212
C04991=1226.859,364.210,-74.759,-175.862,7.461,148.212
C04992=1226.862,363.963,-74.726,-175.863,7.458,148.212
C04993=1226.867,363.715,-74.693,-175.865,7.455,148.212
C04994=1226.871,363.467,-74.660,-175.866,7.452,148.211
C04995=1226.875,363.219,-74.627,-175.868,7.449,148.211
C04996=1226.879,362.971,-74.595,-175.869,7.446,148.211
C04997=1226.884,362.724,-74.563,-175.871,7.444,148.210
C04998=1226.888,362.476,-74.529,-175.872,7.441,148.210
C04999=1226.892,362.228,-74.497,-175.873,7.438,148.210
C05000=1226.896,361.980,-74.464,-175.875,7.436,148.210
C05001=1226.900,361.732,-74.432,-175.877,7.433,148.210
C05002=1226.904,361.484,-74.399,-175.878,7.430,148.209
C05003=1226.908,361.237,-74.366,-175.880,7.427,148.209
C05004=1226.912,360.989,-74.334,-175.882,7.425,148.209
C05005=1226.917,360.742,-74.301,-175.883,7.422,148.208
C05006=1226.921,360.493,-74.269,-175.884,7.419,148.208
C05007=1226.925,360.246,-74.236,-175.886,7.417,148.208
C05008=1226.929,359.997,-74.204,-175.888,7.413,148.207
C05009=1226.933,359.750,-74.170,-175.889,7.410,148.207
C05010=1226.938,359.501,-74.138,-175.891,7.408,148.207
C05011=1226.941,359.254,-74.105,-175.892,7.405,148.207
C05012=1226.946,359.006,-74.073,-175.894,7.403,148.207
C05013=1226.950,358.759,-74.040,-175.896,7.400,148.206
C05014=1226.954,358.510,-74.008,-175.897,7.396,148.206
C05015=1226.958,358.262,-73.976,-175.899,7.394,148.206
C05016=1226.962,358.015,-73.943,-175.900,7.391,148.206
C05017=1226.966,357.766,-73.911,-175.902,7.389,148.205
C05018=1226.971,357.519,-73.878,-175.903,7.386,148.205
C05019=1226.975,357.271,-73.846,-175.905,7.383,148.205
C05020=1226.979,357.024,-73.813,-175.907,7.380,148.205
C05021=1226.983,356.775,-73.781,-175.909,7.378,148.204
C05022=1226.987,356.527,-73.749,-175.910,7.375,148.204
C05023=1226.992,356.280,-73.716,-175.911,7.372,148.204
C05024=1226.995,356.032,-73.684,-175.913,7.370,148.204
C05025=1227.000,355.784,-73.652,-175.915,7.366,148.203
C05026=1227.004,355.536,-73.619,-175.917,7.364,148.203
C05027=1227.008,355.288,-73.587,-175.919,7.361,148.203
C05028=1227.013,355.040,-73.555,-175.920,7.358,148.203
C05029=1227.016,354.793,-73.522,-175.921,7.356,148.202
C05030=1227.021,354.545,-73.490,-175.924,7.353,148.202
C05031=1227.024,354.297,-73.458,-175.925,7.350,148.202
C05032=1227.029,354.049,-73.426,-175.927,7.347,148.202
C05033=1227.033,353.801,-73.393,-175.928,7.345,148.202
C05034=1227.037,353.553,-73.361,-175.930,7.342,148.201
C05035=1227.042,353.305,-73.328,-175.932,7.339,148.201
C05036=1227.046,353.057,-73.297,-175.933,7.336,148.201
C05037=1227.050,352.810,-73.264,-175.935,7.334,148.201
C05038=1227.054,352.562,-73.232,-175.937,7.331,148.200
C05039=1227.058,352.313,-73.199,-175.939,7.328,148.200
C05040=1227.062,352.066,-73.168,-175.940,7.325,148.200
C05041=1227.067,351.818,-73.135,-175.942,7.323,148.200
C05042=1227.070,351.570,-73.103,-175.944,7.320,148.200
C05043=1227.075,351.322,-73.070,-175.945,7.318,148.199
C05044=1227.079,351.075,-73.039,-175.948,7.314,148.199
C05045=1227.083,350.826,-73.007,-175.949,7.312,148.199
C05046=1227.087,350.578,-72.975,-175.951,7.309,148.199
C05047=1227.092,350.331,-72.943,-175.952,7.307,148.199
C05048=1227.096,350.082,-72.911,-175.955,7.303,148.198
C05049=1227.100,349.834,-72.879,-175.956,7.301,148.198
C05050=1227.105,349.587,-72.847,-175.958,7.298,148.198
C05051=1227.108,349.339,-72.814,-175.959,7.296,148.198
C05052=1227.113,349.091,-72.782,-175.962,7.292,148.198
C05053=1227.117,348.844,-72.750,-175.963,7.290,148.197
C05054=1227.121,348.596,-72.719,-175.965,7.287,148.197
C05055=1227.125,348.347,-72.686,-175.967,7.285,148.197
C05056=1227.129,348.100,-72.655,-175.969,7.281,148.197
C05057=1227.134,347.852,-72.622,-175.970,7.279,148.197
C05058=1227.137,347.604,-72.590,-175.972,7.276,148.197
C05059=1227.142,347.356,-72.559,-175.974,7.274,148.196
C05060=1227.146,347.108,-72.526,-175.976,7.270,148.196
C05061=1227.150,346.860,-72.495,-175.977,7.268,148.196
C05062=1227.154,346.612,-72.463,-175.979,7.265,148.196
C05063=1227.159,346.364,-72.431,-175.982,7.262,148.196
C05064=1227.162,346.116,-72.399,-175.983,7.260,148.196
C05065=1227.167,345.868,-72.368,-175.985,7.257,148.195
C05066=1227.171,345.620,-72.336,-175.987,7.255,148.195
C05067=1227.175,345.372,-72.304,-175.989,7.251,148.195
C05068=1227.179,345.124,-72.272,-175.990,7.249,148.195
C05069=1227.184,344.876,-72.240,-175.992,7.246,148.195
C05070=1227.188,344.629,-72.208,-175.994,7.244,148.194
C05071=1227.192,344.381,-72.177,-175.996,7.241,148.194
C05072=1227.196,344.132,-72.144,-175.998,7.238,148.194
C05073=1227.201,343.884,-72.113,-176.000,7.236,148.194
C05074=1227.205,343.636,-72.081,-176.002,7.232,148.194
C05075=1227.209,343.389,-72.050,-176.003,7.230,148.194
C05076=1227.213,343.141,-72.018,-176.005,7.228,148.194
C05077=1227.218,342.893,-71.986,-176.007,7.225,148.193
C05078=1227.222,342.645,-71.955,-176.009,7.222,148.193
C05079=1227.225,342.397,-71.923,-176.011,7.219,148.193
C05080=1227.231,342.149,-71.891,-176.012,7.217,148.193
C05081=1227.234,341.901,-71.859,-176.015,7.214,148.193
C05082=1227.239,341.623,-71.824,-176.017,7.211,148.193
C05083=1227.244,341.346,-71.789,-176.019,7.208,148.192
C05084=1227.248,341.068,-71.753,-176.021,7.204,148.192
C05085=1227.253,340.790,-71.718,-176.023,7.202,148.192
C05086=1227.258,340.543,-71.686,-176.025,7.199,148.192
C05087=1227.261,340.295,-71.655,-176.027,7.196,148.192
C05088=1227.266,340.047,-71.624,-176.029,7.194,148.192
C05089=1227.270,339.799,-71.592,-176.031,7.191,148.192
C05090=1227.273,339.551,-71.560,-176.033,7.188,148.191
C05091=1227.279,339.302,-71.529,-176.035,7.186,148.191
C05092=1227.283,339.054,-71.497,-176.037,7.183,148.191
C05093=1227.287,338.807,-71.465,-176.039,7.180,148.191
C05094=1227.291,338.558,-71.434,-176.040,7.177,148.191
C05095=1227.295,338.311,-71.403,-176.043,7.175,148.191
C05096=1227.299,338.062,-71.372,-176.045,7.172,148.191
C05097=1227.303,337.815,-71.340,-176.046,7.169,148.191
C05098=1227.307,337.567,-71.308,-176.048,7.167,148.191
C05099=1227.312,337.319,-71.278,-176.050,7.165,148.190
C05100=1227.316,337.071,-71.245,-176.052,7.161,148.190
C05101=1227.321,336.823,-71.214,-176.054,7.159,148.190
C05102=1227.325,336.575,-71.183,-176.056,7.156,148.190
C05103=1227.329,336.327,-71.152,-176.058,7.153,148.190
C05104=1227.333,336.079,-71.120,-176.060,7.151,148.190
C05105=1227.338,335.831,-71.089,-176.062,7.148,148.190
C05106=1227.341,335.583,-71.057,-176.065,7.145,148.190
C05107=1227.346,335.335,-71.027,-176.066,7.143,148.189
C05108=1227.350,335.087,-70.995,-176.068,7.140,148.189
C05109=1227.354,334.839,-70.964,-176.070,7.137,148.189
C05110=1227.358,334.591,-70.933,-176.072,7.135,148.189
C05111=1227.362,334.343,-70.901,-176.074,7.132,148.189
C05112=1227.367,334.095,-70.871,-176.076,7.130,148.189
C05113=1227.371,333.847,-70.839,-176.078,7.126,148.189
C05114=1227.375,333.599,-70.808,-176.080,7.124,148.189
C05115=1227.379,333.351,-70.776,-176.082,7.122,148.189
C05116=1227.384,333.103,-70.745,-176.084,7.119,148.189
C05117=1227.388,332.855,-70.715,-176.086,7.116,148.188
C05118=1227.392,332.607,-70.683,-176.088,7.114,148.188
C05119=1227.397,332.359,-70.652,-176.090,7.111,148.188
C05120=1227.401,332.110,-70.621,-176.092,7.108,148.188
C05121=1227.405,331.863,-70.589,-176.094,7.106,148.188
C05122=1227.410,331.615,-70.559,-176.097,7.103,148.188
C05123=1227.414,331.366,-70.528,-176.098,7.100,148.188
C05124=1227.417,331.119,-70.497,-176.100,7.098,148.188
C05125=1227.421,330.870,-70.466,-176.103,7.095,148.188
C05126=1227.426,330.622,-70.435,-176.105,7.092,148.188
C05127=1227.430,330.374,-70.404,-176.106,7.090,148.188
C05128=1227.434,330.126,-70.372,-176.109,7.087,148.188
C05129=1227.439,329.878,-70.341,-176.111,7.084,148.187
C05130=1227.443,329.631,-70.311,-176.113,7.082,148.187
C05131=1227.447,329.382,-70.280,-176.115,7.079,148.187
C05132=1227.452,329.134,-70.249,-176.117,7.076,148.187
C05133=1227.456,328.887,-70.218,-176.119,7.074,148.187
C05134=1227.460,328.638,-70.187,-176.121,7.072,148.187
C05135=1227.464,328.390,-70.156,-176.123,7.069,148.187
C05136=1227.468,328.142,-70.125,-176.125,7.066,148.187
C05137=1227.473,327.894,-70.094,-176.127,7.064,148.187
C05138=1227.477,327.646,-70.063,-176.129,7.060,148.187
C05139=1227.481,327.398,-70.033,-176.131,7.058,148.187
C05140=1227.485,327.150,-70.001,-176.133,7.056,148.187
C05141=1227.490,326.902,-69.971,-176.136,7.053,148.187
C05142=1227.494,326.654,-69.940,-176.138,7.050,148.187
C05143=1227.498,326.405,-69.909,-176.140,7.048,148.187
C05144=1227.502,326.158,-69.878,-176.142,7.045,148.186
C05145=1227.507,325.910,-69.848,-176.144,7.043,148.187
C05146=1227.511,325.661,-69.817,-176.146,7.040,148.186
C05147=1227.515,325.413,-69.786,-176.148,7.037,148.186
C05148=1227.519,325.166,-69.756,-176.150,7.035,148.186
C05149=1227.523,324.917,-69.725,-176.152,7.032,148.186
C05150=1227.528,324.669,-69.694,-176.155,7.029,148.186
C05151=1227.532,324.421,-69.664,-176.157,7.027,148.186
C05152=1227.536,324.173,-69.633,-176.158,7.024,148.186
C05153=1227.540,323.925,-69.602,-176.161,7.021,148.186
C05154=1227.545,323.677,-69.571,-176.163,7.019,148.186
C05155=1227.549,323.429,-69.541,-176.165,7.017,148.186
C05156=1227.553,323.181,-69.510,-176.167,7.014,148.186
C05157=1227.557,322.932,-69.479,-176.170,7.011,148.186
C05158=1227.561,322.685,-69.449,-176.172,7.009,148.186
C05159=1227.566,322.437,-69.418,-176.174,7.006,148.186
C05160=1227.571,322.188,-69.388,-176.176,7.004,148.186
C05161=1227.574,321.940,-69.357,-176.178,7.001,148.186
C05162=1227.579,321.692,-69.327,-176.180,6.998,148.186
C05163=1227.583,321.444,-69.296,-176.182,6.996,148.186
C05164=1227.587,321.196,-69.266,-176.184,6.994,148.186
C05165=1227.591,320.948,-69.235,-176.187,6.990,148.186
C05166=1227.595,320.700,-69.204,-176.189,6.988,148.186
C05167=1227.600,320.451,-69.174,-176.191,6.986,148.186
C05168=1227.605,320.204,-69.144,-176.193,6.983,148.186
C05169=1227.609,319.956,-69.113,-176.196,6.980,148.186
C05170=1227.613,319.707,-69.082,-176.197,6.978,148.186
C05171=1227.617,319.459,-69.053,-176.200,6.975,148.185
C05172=1227.621,319.211,-69.022,-176.202,6.973,148.186
C05173=1227.625,318.963,-68.992,-176.204,6.970,148.186
C05174=1227.630,318.715,-68.961,-176.206,6.968,148.186
C05175=1227.633,318.466,-68.931,-176.208,6.965,148.185
C05176=1227.638,318.218,-68.900,-176.210,6.963,148.185
C05177=1227.643,317.971,-68.870,-176.213,6.960,148.186
C05178=1227.647,317.722,-68.840,-176.215,6.957,148.186
C05179=1227.651,317.474,-68.810,-176.217,6.955,148.186
C05180=1227.655,317.227,-68.779,-176.219,6.953,148.185
C05181=1227.660,316.977,-68.749,-176.222,6.950,148.185
C05182=1227.664,316.730,-68.719,-176.224,6.947,148.185
C05183=1227.668,316.482,-68.688,-176.226,6.945,148.185
C05184=1227.672,316.233,-68.659,-176.228,6.942,148.185
C05185=1227.677,315.986,-68.628,-176.231,6.940,148.186
C05186=1227.681,315.709,-68.595,-176.233,6.937,148.186
C05187=1227.686,315.434,-68.561,-176.235,6.934,148.186
C05188=1227.691,315.158,-68.528,-176.238,6.931,148.186
C05189=1227.696,314.882,-68.494,-176.240,6.928,148.185
C05190=1227.700,314.634,-68.464,-176.242,6.926,148.185
C05191=1227.705,314.386,-68.433,-176.244,6.924,148.185
C05192=1227.709,314.138,-68.404,-176.247,6.921,148.185
C05193=1227.713,313.890,-68.374,-176.249,6.918,148.185
C05194=1227.718,313.642,-68.344,-176.251,6.916,148.186
C05195=1227.721,313.393,-68.313,-176.254,6.913,148.186
C05196=1227.726,313.145,-68.283,-176.256,6.911,148.186
C05197=1227.730,312.897,-68.253,-176.258,6.909,148.186
C05198=1227.734,312.649,-68.224,-176.261,6.906,148.186
C05199=1227.738,312.401,-68.193,-176.262,6.903,148.185
C05200=1227.743,312.153,-68.163,-176.264,6.901,148.186
C05201=1227.746,311.905,-68.133,-176.267,6.898,148.186
C05202=1227.751,311.656,-68.103,-176.269,6.896,148.186
C05203=1227.756,311.408,-68.074,-176.271,6.893,148.186
C05204=1227.759,311.161,-68.044,-176.274,6.890,148.186
C05205=1227.764,310.912,-68.013,-176.276,6.888,148.186
C05206=1227.768,310.664,-67.983,-176.278,6.886,148.186
C05207=1227.772,310.416,-67.954,-176.280,6.884,148.186
C05208=1227.777,310.167,-67.924,-176.283,6.881,148.186
C05209=1227.781,309.920,-67.894,-176.285,6.878,148.186
C05210=1227.785,309.672,-67.864,-176.287,6.876,148.186
C05211=1227.790,309.423,-67.834,-176.290,6.873,148.186
C05212=1227.794,309.175,-67.805,-176.292,6.871,148.186
C05213=1227.798,308.927,-67.774,-176.294,6.869,148.186
C05214=1227.803,308.679,-67.745,-176.297,6.866,148.186
C05215=1227.807,308.430,-67.715,-176.299,6.863,148.186
C05216=1227.811,308.183,-67.685,-176.301,6.861,148.186
C05217=1227.816,307.934,-67.655,-176.303,6.858,148.186
C05218=1227.820,307.686,-67.626,-176.306,6.856,148.186
C05219=1227.825,307.437,-67.596,-176.308,6.854,148.186
C05220=1227.829,307.189,-67.566,-176.310,6.851,148.186
C05221=1227.833,306.942,-67.536,-176.312,6.848,148.186
C05222=1227.837,306.693,-67.507,-176.315,6.846,148.186
C05223=1227.842,306.445,-67.477,-176.317,6.844,148.186
C05224=1227.846,306.196,-67.447,-176.319,6.841,148.186
C05225=1227.850,305.948,-67.418,-176.321,6.839,148.186
C05226=1227.854,305.700,-67.388,-176.324,6.836,148.186
C05227=1227.859,305.452,-67.359,-176.326,6.833,148.186
C05228=1227.862,305.204,-67.329,-176.328,6.831,148.187
C05229=1227.867,304.955,-67.299,-176.330,6.829,148.187
C05230=1227.871,304.707,-67.269,-176.332,6.827,148.187
C05231=1227.876,304.459,-67.240,-176.336,6.824,148.187
C05232=1227.880,304.211,-67.211,-176.338,6.822,148.187
C05233=1227.885,303.963,-67.181,-176.340,6.819,148.187
C05234=1227.889,303.715,-67.152,-176.342,6.816,148.187
C05235=1227.893,303.467,-67.122,-176.345,6.814,148.187
C05236=1227.897,303.218,-67.093,-176.347,6.812,148.187
C05237=1227.902,302.970,-67.063,-176.349,6.810,148.187
C05238=1227.906,302.721,-67.033,-176.351,6.807,148.187
C05239=1227.910,302.473,-67.004,-176.354,6.804,148.187
C05240=1227.915,302.225,-66.974,-176.356,6.802,148.187
C05241=1227.919,301.977,-66.945,-176.359,6.800,148.187
C05242=1227.924,301.729,-66.916,-176.361,6.797,148.188
C05243=1227.928,301.481,-66.887,-176.363,6.795,148.188
C05244=1227.932,301.232,-66.857,-176.365,6.793,148.188
C05245=1227.936,300.984,-66.828,-176.368,6.790,148.188
C05246=1227.940,300.736,-66.798,-176.370,6.788,148.188
C05247=1227.945,300.488,-66.769,-176.372,6.785,148.188
C05248=1227.949,300.239,-66.740,-176.375,6.782,148.188
C05249=1227.954,299.991,-66.711,-176.377,6.780,148.188
C05250=1227.958,299.743,-66.681,-176.379,6.778,148.188
C05251=1227.962,299.495,-66.652,-176.381,6.776,148.188
C05252=1227.966,299.246,-66.623,-176.384,6.773,148.188
C05253=1227.970,298.998,-66.593,-176.386,6.771,148.188
C05254=1227.975,298.749,-66.564,-176.388,6.768,148.188
C05255=1227.980,298.502,-66.535,-176.391,6.766,148.189
C05256=1227.984,298.253,-66.506,-176.394,6.764,148.189
C05257=1227.988,298.005,-66.476,-176.396,6.761,148.189
C05258=1227.992,297.757,-66.447,-176.398,6.759,148.189
C05259=1227.997,297.508,-66.418,-176.400,6.756,148.189
C05260=1228.002,297.260,-66.389,-176.403,6.754,148.189
C05261=1228.006,297.012,-66.360,-176.405,6.752,148.189
C05262=1228.009,296.764,-66.331,-176.407,6.750,148.189
C05263=1228.014,296.515,-66.302,-176.410,6.747,148.189
C05264=1228.018,296.267,-66.273,-176.412,6.744,148.189
C05265=1228.023,296.020,-66.243,-176.415,6.742,148.189
C05266=1228.027,295.771,-66.215,-176.417,6.740,148.190
C05267=1228.031,295.522,-66.185,-176.419,6.737,148.190
C05268=1228.036,295.274,-66.156,-176.421,6.735,148.190
C05269=1228.041,295.026,-66.127,-176.424,6.733,148.190
C05270=1228.044,294.778,-66.099,-176.427,6.730,148.190
C05271=1228.048,294.530,-66.069,-176.429,6.728,148.190
C05272=1228.053,294.281,-66.040,-176.431,6.726,148.190
C05273=1228.057,294.033,-66.011,-176.433,6.723,148.190
C05274=1228.062,293.784,-65.983,-176.436,6.721,148.190
C05275=1228.066,293.536,-65.953,-176.438,6.718,148.190
C05276=1228.070,293.288,-65.924,-176.440,6.716,148.190
C05277=1228.075,293.040,-65.896,-176.443,6.714,148.191
C05278=1228.079,292.792,-65.866,-176.446,6.711,148.191
C05279=1228.083,292.543,-65.838,-176.448,6.709,148.191
C05280=1228.087,292.295,-65.809,-176.450,6.707,148.191
C05281=1228.092,292.047,-65.780,-176.452,6.705,148.191
C05282=1228.096,291.798,-65.751,-176.455,6.702,148.191
C05283=1228.101,291.549,-65.722,-176.457,6.700,148.191
C05284=1228.105,291.302,-65.694,-176.459,6.697,148.191
C05285=1228.109,291.053,-65.665,-176.462,6.696,148.192
C05286=1228.113,290.805,-65.636,-176.465,6.692,148.192
C05287=1228.118,290.557,-65.607,-176.467,6.690,148.192
C05288=1228.122,290.308,-65.579,-176.469,6.688,148.192
C05289=1228.126,290.060,-65.550,-176.471,6.686,148.192
C05290=1228.131,289.786,-65.518,-176.474,6.683,148.192
C05291=1228.137,289.512,-65.487,-176.477,6.681,148.192
C05292=1228.141,289.238,-65.455,-176.479,6.678,148.192
C05293=1228.146,288.964,-65.423,-176.482,6.675,148.192
C05294=1228.150,288.715,-65.395,-176.485,6.673,148.193
C05295=1228.155,288.467,-65.366,-176.487,6.671,148.193
C05296=1228.159,288.219,-65.337,-176.489,6.669,148.193
C05297=1228.163,287.970,-65.309,-176.491,6.667,148.193
C05298=1228.168,287.722,-65.280,-176.494,6.664,148.193
C05299=1228.172,287.474,-65.251,-176.497,6.662,148.193
C05300=1228.176,287.226,-65.223,-176.499,6.660,148.193
C05301=1228.181,286.977,-65.194,-176.501,6.658,148.194
C05302=1228.185,286.728,-65.166,-176.504,6.655,148.194
C05303=1228.189,286.481,-65.137,-176.506,6.653,148.194
C05304=1228.194,286.232,-65.108,-176.509,6.651,148.194
C05305=1228.198,285.984,-65.081,-176.511,6.648,148.194
C05306=1228.203,285.735,-65.052,-176.513,6.646,148.194
C05307=1228.206,285.487,-65.023,-176.516,6.643,148.194
C05308=1228.211,285.239,-64.995,-176.518,6.641,148.194
C05309=1228.216,284.990,-64.966,-176.520,6.639,148.194
C05310=1228.220,284.742,-64.938,-176.523,6.637,148.195
C05311=1228.224,284.494,-64.909,-176.525,6.635,148.195
C05312=1228.229,284.246,-64.882,-176.528,6.632,148.195
C05313=1228.233,283.997,-64.852,-176.530,6.630,148.195
C05314=1228.237,283.749,-64.824,-176.532,6.628,148.195
C05315=1228.242,283.501,-64.796,-176.535,6.626,148.195
C05316=1228.246,283.252,-64.767,-176.537,6.624,148.196
C05317=1228.251,283.004,-64.739,-176.540,6.621,148.196
C05318=1228.254,282.755,-64.711,-176.542,6.619,148.196
C05319=1228.259,282.507,-64.683,-176.544,6.616,148.196
C05320=1228.263,282.258,-64.654,-176.547,6.615,148.196
C05321=1228.268,282.010,-64.626,-176.549,6.612,148.196
C05322=1228.272,281.762,-64.598,-176.552,6.610,148.197
C05323=1228.277,281.514,-64.569,-176.554,6.607,148.197
C05324=1228.281,281.265,-64.541,-176.557,6.605,148.197
C05325=1228.285,281.017,-64.514,-176.559,6.603,148.197
C05326=1228.290,280.768,-64.485,-176.561,6.601,148.197
C05327=1228.294,280.520,-64.457,-176.564,6.598,148.197
C05328=1228.299,280.271,-64.428,-176.567,6.596,148.197
C05329=1228.303,280.024,-64.401,-176.569,6.594,148.198
C05330=1228.307,279.775,-64.372,-176.571,6.592,148.198
C05331=1228.312,279.527,-64.344,-176.574,6.590,148.198
C05332=1228.315,279.278,-64.316,-176.576,6.587,148.198
C05333=1228.321,279.030,-64.288,-176.579,6.585,148.198
C05334=1228.324,278.781,-64.259,-176.581,6.583,148.198
C05335=1228.329,278.534,-64.232,-176.583,6.581,148.198
C05336=1228.333,278.285,-64.203,-176.586,6.579,148.199
C05337=1228.338,278.037,-64.175,-176.588,6.577,148.199
C05338=1228.342,277.788,-64.148,-176.591,6.574,148.199
C05339=1228.347,277.539,-64.119,-176.593,6.572,148.199
C05340=1228.351,277.292,-64.091,-176.596,6.570,148.199
C05341=1228.355,277.043,-64.063,-176.598,6.568,148.199
C05342=1228.360,276.795,-64.035,-176.601,6.566,148.200
C05343=1228.364,276.546,-64.007,-176.603,6.563,148.200
C05344=1228.368,276.298,-63.980,-176.606,6.561,148.200
C05345=1228.373,276.049,-63.951,-176.608,6.558,148.200
C05346=1228.377,275.801,-63.923,-176.611,6.557,148.200
C05347=1228.381,275.553,-63.895,-176.613,6.554,148.201
C05348=1228.386,275.304,-63.868,-176.615,6.552,148.201
C05349=1228.391,275.056,-63.840,-176.617,6.550,148.201
C05350=1228.394,274.807,-63.812,-176.621,6.548,148.201
C05351=1228.399,274.559,-63.784,-176.623,6.545,148.201
C05352=1228.403,274.311,-63.757,-176.625,6.543,148.201
C05353=1228.408,274.062,-63.728,-176.627,6.541,148.202
C05354=1228.412,273.814,-63.700,-176.630,6.539,148.202
C05355=1228.416,273.565,-63.673,-176.632,6.537,148.202
C05356=1228.421,273.317,-63.645,-176.635,6.535,148.202
C05357=1228.425,273.069,-63.617,-176.637,6.532,148.202
C05358=1228.430,272.820,-63.589,-176.640,6.530,148.203
C05359=1228.434,272.572,-63.561,-176.643,6.528,148.203
C05360=1228.439,272.323,-63.534,-176.645,6.526,148.203
C05361=1228.442,272.075,-63.506,-176.647,6.524,148.203
C05362=1228.447,271.827,-63.478,-176.649,6.522,148.203
C05363=1228.452,271.578,-63.451,-176.652,6.520,148.204
C05364=1228.456,271.329,-63.423,-176.655,6.517,148.204
C05365=1228.461,271.081,-63.396,-176.657,6.515,148.204
C05366=1228.465,270.833,-63.368,-176.659,6.513,148.204
C05367=1228.469,270.584,-63.340,-176.662,6.511,148.204
C05368=1228.473,270.336,-63.313,-176.664,6.509,148.204
C05369=1228.478,270.087,-63.286,-176.667,6.507,148.205
C05370=1228.482,269.839,-63.257,-176.669,6.505,148.205
C05371=1228.487,269.590,-63.230,-176.671,6.503,148.205
C05372=1228.492,269.342,-63.202,-176.675,6.500,148.205
C05373=1228.496,269.094,-63.175,-176.677,6.498,148.205
C05374=1228.500,268.845,-63.147,-176.679,6.496,148.206
C05375=1228.505,268.597,-63.120,-176.681,6.494,148.206
C05376=1228.509,268.349,-63.092,-176.684,6.492,148.206
C05377=1228.513,268.100,-63.064,-176.687,6.490,148.206
C05378=1228.518,267.851,-63.037,-176.689,6.488,148.206
C05379=1228.522,267.603,-63.010,-176.691,6.486,148.207
C05380=1228.527,267.355,-62.983,-176.694,6.483,148.207
C05381=1228.530,267.106,-62.954,-176.697,6.481,148.207
C05382=1228.535,266.858,-62.927,-176.699,6.479,148.207
C05383=1228.540,266.609,-62.900,-176.701,6.477,148.207
C05384=1228.544,266.361,-62.873,-176.704,6.475,148.208
C05385=1228.548,266.112,-62.845,-176.706,6.473,148.208
C05386=1228.553,265.864,-62.818,-176.709,6.471,148.208
C05387=1228.557,265.616,-62.790,-176.711,6.469,148.208
C05388=1228.562,265.367,-62.763,-176.713,6.467,148.208
C05389=1228.566,265.119,-62.736,-176.716,6.465,148.209
C05390=1228.571,264.869,-62.709,-176.719,6.462,148.209
C05391=1228.575,264.622,-62.681,-176.721,6.460,148.209
C05392=1228.580,264.373,-62.654,-176.724,6.458,148.209
C05393=1228.584,264.125,-62.627,-176.726,6.456,148.209
C05394=1228.589,263.852,-62.597,-176.729,6.454,148.210
C05395=1228.593,263.579,-62.566,-176.732,6.451,148.210
C05396=1228.598,263.307,-62.537,-176.734,6.449,148.210
C05397=1228.603,263.033,-62.507,-176.737,6.448,148.211
C05398=1228.608,262.786,-62.479,-176.740,6.444,148.211
C05399=1228.612,262.537,-62.453,-176.742,6.443,148.211
C05400=1228.616,262.289,-62.426,-176.744,6.440,148.211
C05401=1228.621,262.040,-62.399,-176.747,6.439,148.211
C05402=1228.625,261.791,-62.371,-176.750,6.437,148.212
C05403=1228.630,261.543,-62.344,-176.752,6.434,148.212
C05404=1228.634,261.294,-62.317,-176.754,6.433,148.212
C05405=1228.639,261.046,-62.289,-176.757,6.431,148.212
C05406=1228.643,260.798,-62.263,-176.759,6.428,148.212
C05407=1228.647,260.550,-62.236,-176.762,6.427,148.213
C05408=1228.652,260.301,-62.209,-176.764,6.425,148.213
C05409=1228.656,260.052,-62.181,-176.766,6.422,148.213
C05410=1228.661,259.803,-62.154,-176.769,6.421,148.213
C05411=1228.665,259.555,-62.128,-176.772,6.419,148.214
C05412=1228.669,259.307,-62.101,-176.774,6.416,148.214
C05413=1228.674,259.058,-62.074,-176.777,6.414,148.214
C05414=1228.679,258.810,-62.047,-176.779,6.412,148.214
C05415=1228.683,258.561,-62.020,-176.782,6.410,148.214
C05416=1228.687,258.313,-61.993,-176.784,6.408,148.215
C05417=1228.692,258.065,-61.966,-176.787,6.406,148.215
C05418=1228.696,257.815,-61.939,-176.789,6.404,148.215
C05419=1228.701,257.567,-61.912,-176.791,6.402,148.215
C05420=1228.704,257.319,-61.885,-176.794,6.400,148.216
C05421=1228.709,257.070,-61.858,-176.797,6.398,148.216
C05422=1228.714,256.822,-61.831,-176.799,6.396,148.216
C05423=1228.719,256.573,-61.805,-176.801,6.394,148.216
C05424=1228.723,256.324,-61.778,-176.804,6.392,148.217
C05425=1228.727,256.076,-61.751,-176.806,6.390,148.217
C05426=1228.732,255.827,-61.724,-176.809,6.388,148.217
C05427=1228.736,255.579,-61.698,-176.811,6.386,148.217
C05428=1228.741,255.331,-61.671,-176.814,6.384,148.218
C05429=1228.745,255.082,-61.643,-176.816,6.382,148.218
C05430=1228.749,254.833,-61.618,-176.819,6.380,148.218
C05431=1228.754,254.585,-61.591,-176.821,6.378,148.218
C05432=1228.759,254.336,-61.564,-176.824,6.375,148.218
C05433=1228.763,254.088,-61.537,-176.827,6.373,148.219
C05434=1228.767,253.840,-61.510,-176.829,6.371,148.219
C05435=1228.772,253.591,-61.484,-176.832,6.369,148.219
C05436=1228.776,253.342,-61.457,-176.834,6.367,148.219
C05437=1228.781,253.094,-61.430,-176.837,6.365,148.220
C05438=1228.785,252.846,-61.404,-176.839,6.363,148.220
C05439=1228.790,252.597,-61.377,-176.842,6.362,148.220
C05440=1228.794,252.348,-61.350,-176.844,6.359,148.220
C05441=1228.798,252.100,-61.324,-176.846,6.358,148.221
C05442=1228.803,251.851,-61.298,-176.849,6.356,148.221
C05443=1228.807,251.603,-61.271,-176.852,6.354,148.221
C05444=1228.812,251.354,-61.244,-176.854,6.352,148.221
C05445=1228.816,251.105,-61.218,-176.856,6.350,148.222
C05446=1228.821,250.857,-61.191,-176.859,6.348,148.222
C05447=1228.825,250.609,-61.165,-176.862,6.346,148.222
C05448=1228.830,250.360,-61.138,-176.864,6.344,148.222
C05449=1228.834,250.111,-61.111,-176.866,6.342,148.223
C05450=1228.838,249.863,-61.085,-176.869,6.340,148.223
C05451=1228.843,249.614,-61.059,-176.872,6.338,148.223
C05452=1228.847,249.366,-61.032,-176.874,6.336,148.223
C05453=1228.852,249.116,-61.006,-176.876,6.334,148.224
C05454=1228.856,248.868,-60.979,-176.879,6.332,148.224
C05455=1228.861,248.619,-60.953,-176.882,6.330,148.224
C05456=1228.865,248.371,-60.926,-176.884,6.328,148.224
C05457=1228.869,248.123,-60.900,-176.886,6.326,148.225
C05458=1228.874,247.874,-60.874,-176.889,6.324,148.225
C05459=1228.878,247.626,-60.848,-176.892,6.322,148.225
C05460=1228.883,247.377,-60.821,-176.894,6.320,148.226
C05461=1228.887,247.129,-60.795,-176.896,6.318,148.226
C05462=1228.892,246.880,-60.768,-176.899,6.316,148.226
C05463=1228.896,246.631,-60.743,-176.901,6.315,148.226
C05464=1228.901,246.382,-60.716,-176.904,6.313,148.227
C05465=1228.905,246.134,-60.690,-176.906,6.310,148.227
C05466=1228.909,245.886,-60.663,-176.909,6.309,148.227
C05467=1228.914,245.636,-60.637,-176.911,6.307,148.227
C05468=1228.919,245.389,-60.611,-176.914,6.305,148.228
